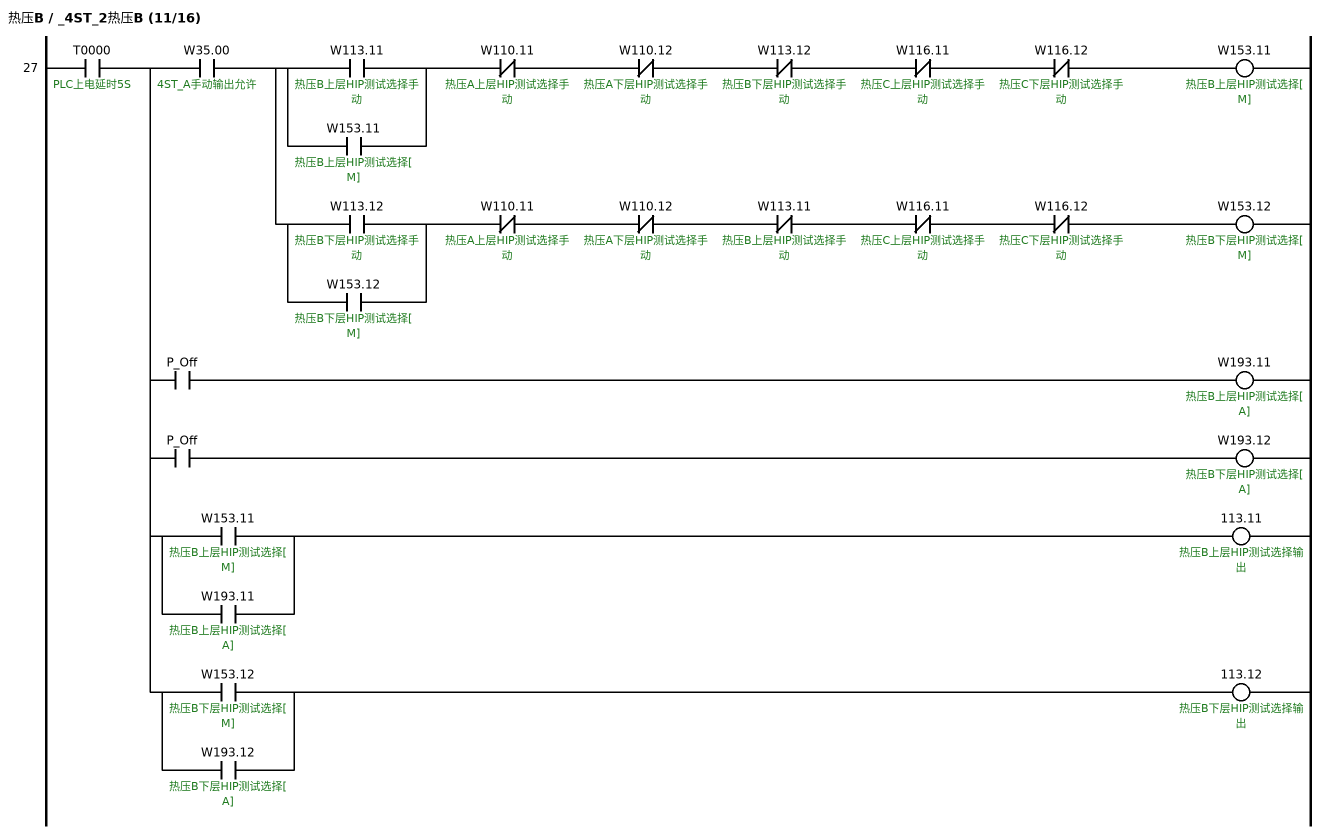
; [picture p192: 热压B / _4ST_2热压B, rungs 27-27]
; rung 27
LD T0000  ; PLC上电延时5S
OUT TR0
AND W35.00  ; 4ST_A手动输出允许
OUT TR1
LD W113.11  ; 热压B上层HIP测试选择手动
OR W153.11  ; 热压B上层HIP测试选择[M]
ANDLD
ANDNOT W110.11  ; 热压A上层HIP测试选择手动
ANDNOT W110.12  ; 热压A下层HIP测试选择手动
ANDNOT W113.12  ; 热压B下层HIP测试选择手动
ANDNOT W116.11  ; 热压C上层HIP测试选择手动
ANDNOT W116.12  ; 热压C下层HIP测试选择手动
OUT W153.11  ; 热压B上层HIP测试选择[M]
LD TR1
LD W113.12  ; 热压B下层HIP测试选择手动
OR W153.12  ; 热压B下层HIP测试选择[M]
ANDLD
ANDNOT W110.11  ; 热压A上层HIP测试选择手动
ANDNOT W110.12  ; 热压A下层HIP测试选择手动
ANDNOT W113.11  ; 热压B上层HIP测试选择手动
ANDNOT W116.11  ; 热压C上层HIP测试选择手动
ANDNOT W116.12  ; 热压C下层HIP测试选择手动
OUT W153.12  ; 热压B下层HIP测试选择[M]
LD TR0
AND P_Off
OUT W193.11  ; 热压B上层HIP测试选择[A]
LD TR0
AND P_Off
OUT W193.12  ; 热压B下层HIP测试选择[A]
LD TR0
LD W153.11  ; 热压B上层HIP测试选择[M]
OR W193.11  ; 热压B上层HIP测试选择[A]
ANDLD
OUT 113.11  ; 热压B上层HIP测试选择输出
LD TR0
LD W153.12  ; 热压B下层HIP测试选择[M]
OR W193.12  ; 热压B下层HIP测试选择[A]
ANDLD
OUT 113.12  ; 热压B下层HIP测试选择输出

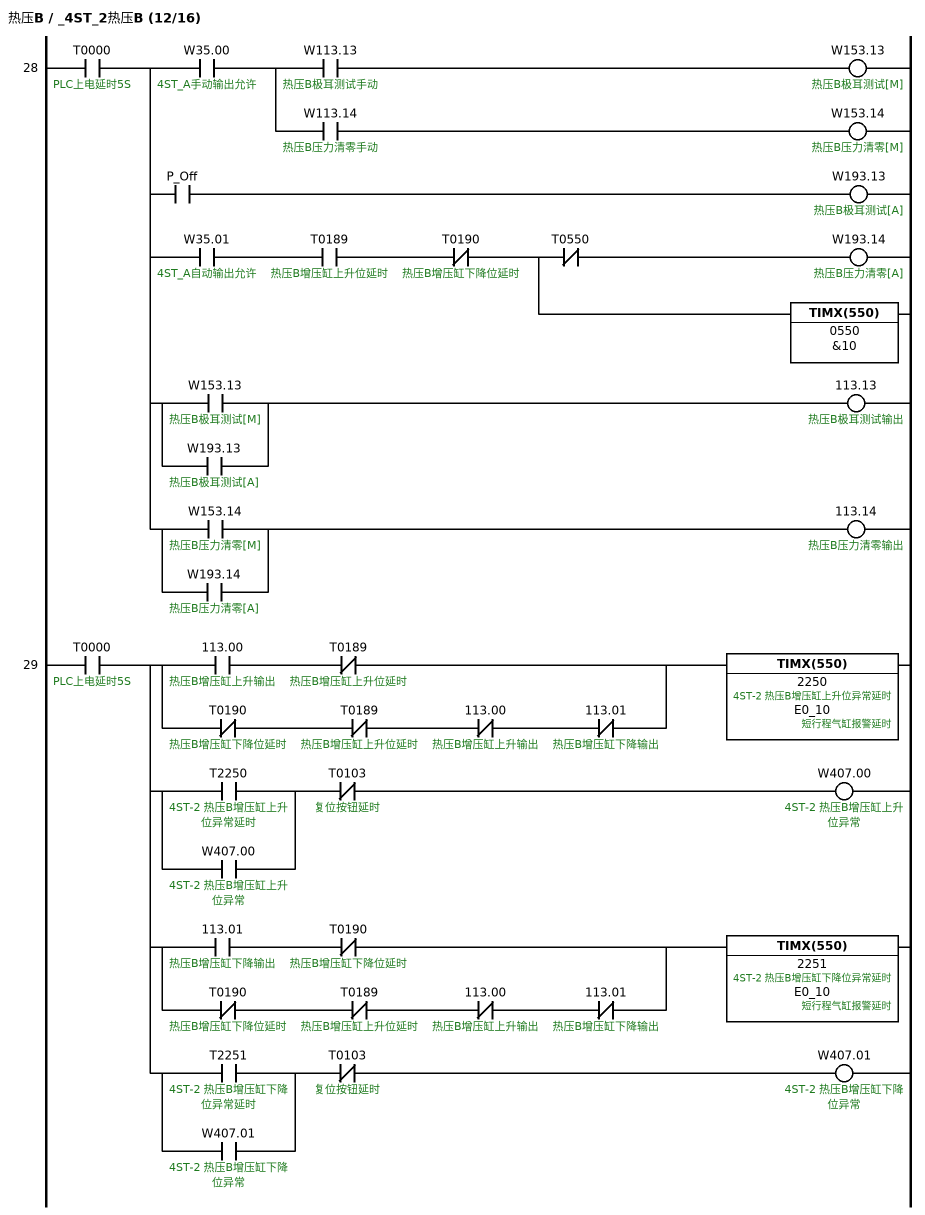
; rung 28
LD T0000  ; PLC上电延时5S
OUT TR0
AND W35.00  ; 4ST_A手动输出允许
OUT TR1
AND W113.13  ; 热压B极耳测试手动
OUT W153.13  ; 热压B极耳测试[M]
LD TR1
AND W113.14  ; 热压B压力清零手动
OUT W153.14  ; 热压B压力清零[M]
LD TR0
AND P_Off
OUT W193.13  ; 热压B极耳测试[A]
LD TR0
AND W35.01  ; 4ST_A自动输出允许
AND T0189  ; 热压B增压缸上升位延时
ANDNOT T0190  ; 热压B增压缸下降位延时
OUT TR1
ANDNOT T0550
OUT W193.14  ; 热压B压力清零[A]
LD TR1
TIMX(550) 0550 &10
LD TR0
LD W153.13  ; 热压B极耳测试[M]
OR W193.13  ; 热压B极耳测试[A]
ANDLD
OUT 113.13  ; 热压B极耳测试输出
LD TR0
LD W153.14  ; 热压B压力清零[M]
OR W193.14  ; 热压B压力清零[A]
ANDLD
OUT 113.14  ; 热压B压力清零输出
; rung 29
LD T0000  ; PLC上电延时5S
OUT TR0
LD 113.00  ; 热压B增压缸上升输出
ANDNOT T0189  ; 热压B增压缸上升位延时
LDNOT T0190  ; 热压B增压缸下降位延时
ANDNOT T0189  ; 热压B增压缸上升位延时
ANDNOT 113.00  ; 热压B增压缸上升输出
ANDNOT 113.01  ; 热压B增压缸下降输出
ORLD
ANDLD
TIMX(550) 2250 E0_10  ; 短行程气缸报警延时, 4ST-2 热压B增压缸上升位异常延时
LD TR0
LD T2250  ; 4ST-2 热压B增压缸上升位异常延时
OR W407.00  ; 4ST-2 热压B增压缸上升位异常
ANDLD
ANDNOT T0103  ; 复位按钮延时
OUT W407.00  ; 4ST-2 热压B增压缸上升位异常
LD TR0
LD 113.01  ; 热压B增压缸下降输出
ANDNOT T0190  ; 热压B增压缸下降位延时
LDNOT T0190  ; 热压B增压缸下降位延时
ANDNOT T0189  ; 热压B增压缸上升位延时
ANDNOT 113.00  ; 热压B增压缸上升输出
ANDNOT 113.01  ; 热压B增压缸下降输出
ORLD
ANDLD
TIMX(550) 2251 E0_10  ; 短行程气缸报警延时, 4ST-2 热压B增压缸下降位异常延时
LD TR0
LD T2251  ; 4ST-2 热压B增压缸下降位异常延时
OR W407.01  ; 4ST-2 热压B增压缸下降位异常
ANDLD
ANDNOT T0103  ; 复位按钮延时
OUT W407.01  ; 4ST-2 热压B增压缸下降位异常

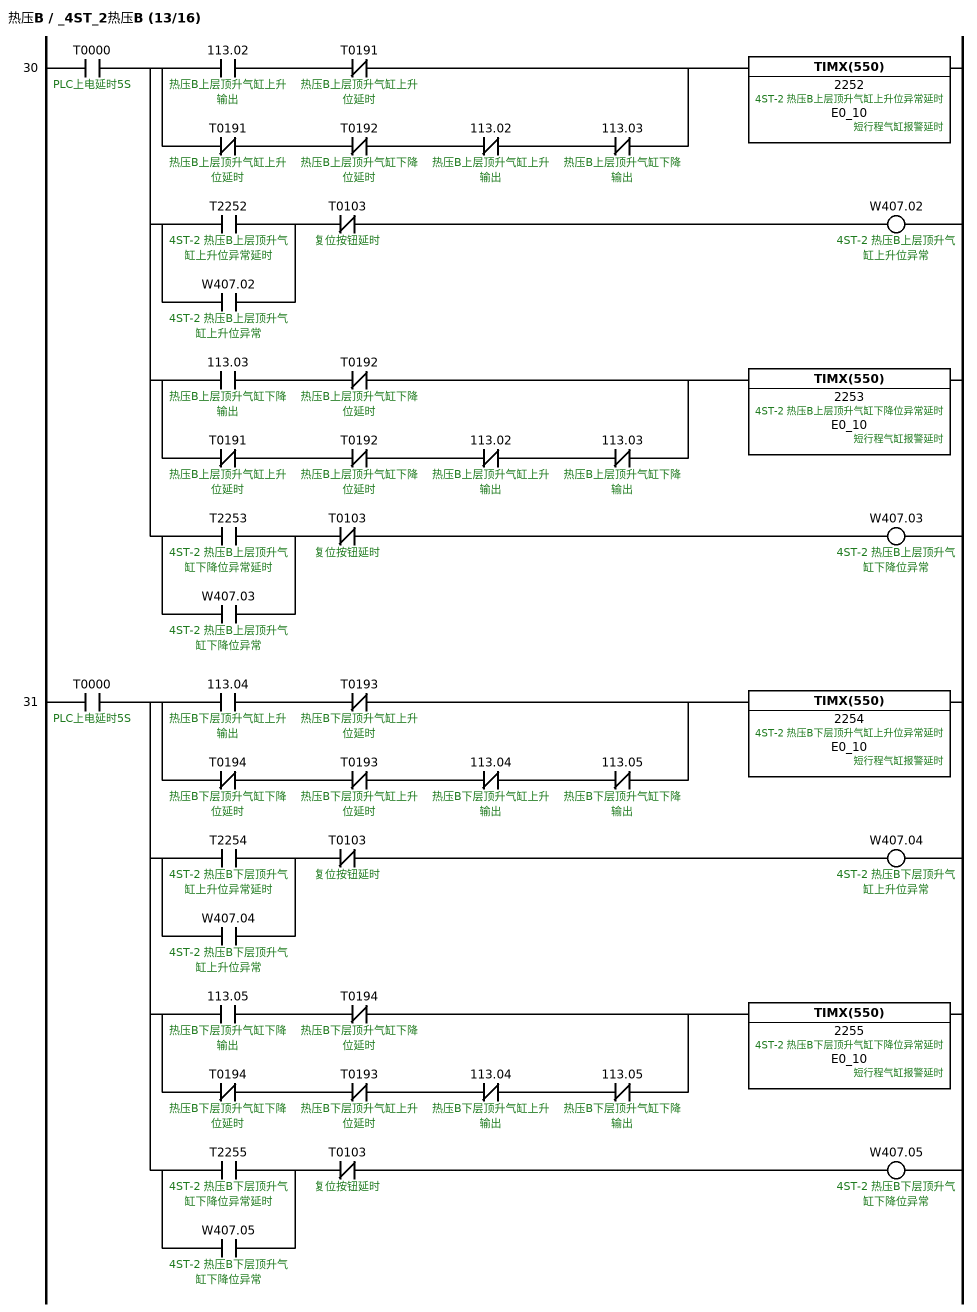
; rung 30
LD T0000  ; PLC上电延时5S
OUT TR0
LD 113.02  ; 热压B上层顶升气缸上升输出
ANDNOT T0191  ; 热压B上层顶升气缸上升位延时
LDNOT T0191  ; 热压B上层顶升气缸上升位延时
ANDNOT T0192  ; 热压B上层顶升气缸下降位延时
ANDNOT 113.02  ; 热压B上层顶升气缸上升输出
ANDNOT 113.03  ; 热压B上层顶升气缸下降输出
ORLD
ANDLD
TIMX(550) 2252 E0_10  ; 短行程气缸报警延时, 4ST-2 热压B上层顶升气缸上升位异常延时
LD TR0
LD T2252  ; 4ST-2 热压B上层顶升气缸上升位异常延时
OR W407.02  ; 4ST-2 热压B上层顶升气缸上升位异常
ANDLD
ANDNOT T0103  ; 复位按钮延时
OUT W407.02  ; 4ST-2 热压B上层顶升气缸上升位异常
LD TR0
LD 113.03  ; 热压B上层顶升气缸下降输出
ANDNOT T0192  ; 热压B上层顶升气缸下降位延时
LDNOT T0191  ; 热压B上层顶升气缸上升位延时
ANDNOT T0192  ; 热压B上层顶升气缸下降位延时
ANDNOT 113.02  ; 热压B上层顶升气缸上升输出
ANDNOT 113.03  ; 热压B上层顶升气缸下降输出
ORLD
ANDLD
TIMX(550) 2253 E0_10  ; 短行程气缸报警延时, 4ST-2 热压B上层顶升气缸下降位异常延时
LD TR0
LD T2253  ; 4ST-2 热压B上层顶升气缸下降位异常延时
OR W407.03  ; 4ST-2 热压B上层顶升气缸下降位异常
ANDLD
ANDNOT T0103  ; 复位按钮延时
OUT W407.03  ; 4ST-2 热压B上层顶升气缸下降位异常
; rung 31
LD T0000  ; PLC上电延时5S
OUT TR0
LD 113.04  ; 热压B下层顶升气缸上升输出
ANDNOT T0193  ; 热压B下层顶升气缸上升位延时
LDNOT T0194  ; 热压B下层顶升气缸下降位延时
ANDNOT T0193  ; 热压B下层顶升气缸上升位延时
ANDNOT 113.04  ; 热压B下层顶升气缸上升输出
ANDNOT 113.05  ; 热压B下层顶升气缸下降输出
ORLD
ANDLD
TIMX(550) 2254 E0_10  ; 短行程气缸报警延时, 4ST-2 热压B下层顶升气缸上升位异常延时
LD TR0
LD T2254  ; 4ST-2 热压B下层顶升气缸上升位异常延时
OR W407.04  ; 4ST-2 热压B下层顶升气缸上升位异常
ANDLD
ANDNOT T0103  ; 复位按钮延时
OUT W407.04  ; 4ST-2 热压B下层顶升气缸上升位异常
LD TR0
LD 113.05  ; 热压B下层顶升气缸下降输出
ANDNOT T0194  ; 热压B下层顶升气缸下降位延时
LDNOT T0194  ; 热压B下层顶升气缸下降位延时
ANDNOT T0193  ; 热压B下层顶升气缸上升位延时
ANDNOT 113.04  ; 热压B下层顶升气缸上升输出
ANDNOT 113.05  ; 热压B下层顶升气缸下降输出
ORLD
ANDLD
TIMX(550) 2255 E0_10  ; 短行程气缸报警延时, 4ST-2 热压B下层顶升气缸下降位异常延时
LD TR0
LD T2255  ; 4ST-2 热压B下层顶升气缸下降位异常延时
OR W407.05  ; 4ST-2 热压B下层顶升气缸下降位异常
ANDLD
ANDNOT T0103  ; 复位按钮延时
OUT W407.05  ; 4ST-2 热压B下层顶升气缸下降位异常

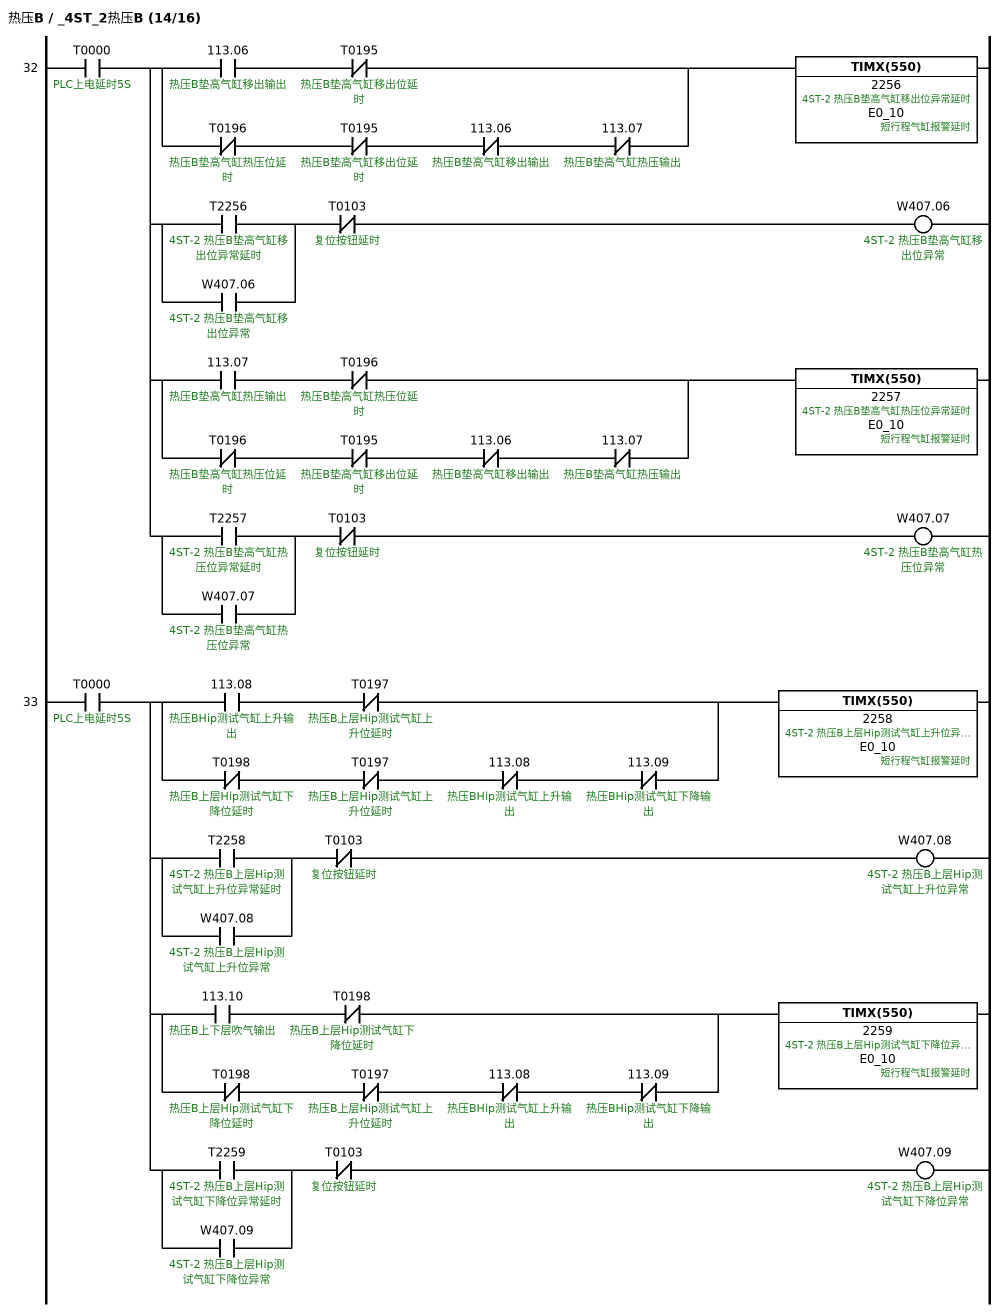
; rung 32
LD T0000  ; PLC上电延时5S
OUT TR0
LD 113.06  ; 热压B垫高气缸移出输出
ANDNOT T0195  ; 热压B垫高气缸移出位延时
LDNOT T0196  ; 热压B垫高气缸热压位延时
ANDNOT T0195  ; 热压B垫高气缸移出位延时
ANDNOT 113.06  ; 热压B垫高气缸移出输出
ANDNOT 113.07  ; 热压B垫高气缸热压输出
ORLD
ANDLD
TIMX(550) 2256 E0_10  ; 短行程气缸报警延时, 4ST-2 热压B垫高气缸移出位异常延时
LD TR0
LD T2256  ; 4ST-2 热压B垫高气缸移出位异常延时
OR W407.06  ; 4ST-2 热压B垫高气缸移出位异常
ANDLD
ANDNOT T0103  ; 复位按钮延时
OUT W407.06  ; 4ST-2 热压B垫高气缸移出位异常
LD TR0
LD 113.07  ; 热压B垫高气缸热压输出
ANDNOT T0196  ; 热压B垫高气缸热压位延时
LDNOT T0196  ; 热压B垫高气缸热压位延时
ANDNOT T0195  ; 热压B垫高气缸移出位延时
ANDNOT 113.06  ; 热压B垫高气缸移出输出
ANDNOT 113.07  ; 热压B垫高气缸热压输出
ORLD
ANDLD
TIMX(550) 2257 E0_10  ; 短行程气缸报警延时, 4ST-2 热压B垫高气缸热压位异常延时
LD TR0
LD T2257  ; 4ST-2 热压B垫高气缸热压位异常延时
OR W407.07  ; 4ST-2 热压B垫高气缸热压位异常
ANDLD
ANDNOT T0103  ; 复位按钮延时
OUT W407.07  ; 4ST-2 热压B垫高气缸热压位异常
; rung 33
LD T0000  ; PLC上电延时5S
OUT TR0
LD 113.08  ; 热压BHip测试气缸上升输出
ANDNOT T0197  ; 热压B上层Hip测试气缸上升位延时
LDNOT T0198  ; 热压B上层Hip测试气缸下降位延时
ANDNOT T0197  ; 热压B上层Hip测试气缸上升位延时
ANDNOT 113.08  ; 热压BHip测试气缸上升输出
ANDNOT 113.09  ; 热压BHip测试气缸下降输出
ORLD
ANDLD
TIMX(550) 2258 E0_10  ; 短行程气缸报警延时, 4ST-2 热压B上层Hip测试气缸上升位异常延时
LD TR0
LD T2258  ; 4ST-2 热压B上层Hip测试气缸上升位异常延时
OR W407.08  ; 4ST-2 热压B上层Hip测试气缸上升位异常
ANDLD
ANDNOT T0103  ; 复位按钮延时
OUT W407.08  ; 4ST-2 热压B上层Hip测试气缸上升位异常
LD TR0
LD 113.10  ; 热压B上下层吹气输出
ANDNOT T0198  ; 热压B上层Hip测试气缸下降位延时
LDNOT T0198  ; 热压B上层Hip测试气缸下降位延时
ANDNOT T0197  ; 热压B上层Hip测试气缸上升位延时
ANDNOT 113.08  ; 热压BHip测试气缸上升输出
ANDNOT 113.09  ; 热压BHip测试气缸下降输出
ORLD
ANDLD
TIMX(550) 2259 E0_10  ; 短行程气缸报警延时, 4ST-2 热压B上层Hip测试气缸下降位异常延时
LD TR0
LD T2259  ; 4ST-2 热压B上层Hip测试气缸下降位异常延时
OR W407.09  ; 4ST-2 热压B上层Hip测试气缸下降位异常
ANDLD
ANDNOT T0103  ; 复位按钮延时
OUT W407.09  ; 4ST-2 热压B上层Hip测试气缸下降位异常

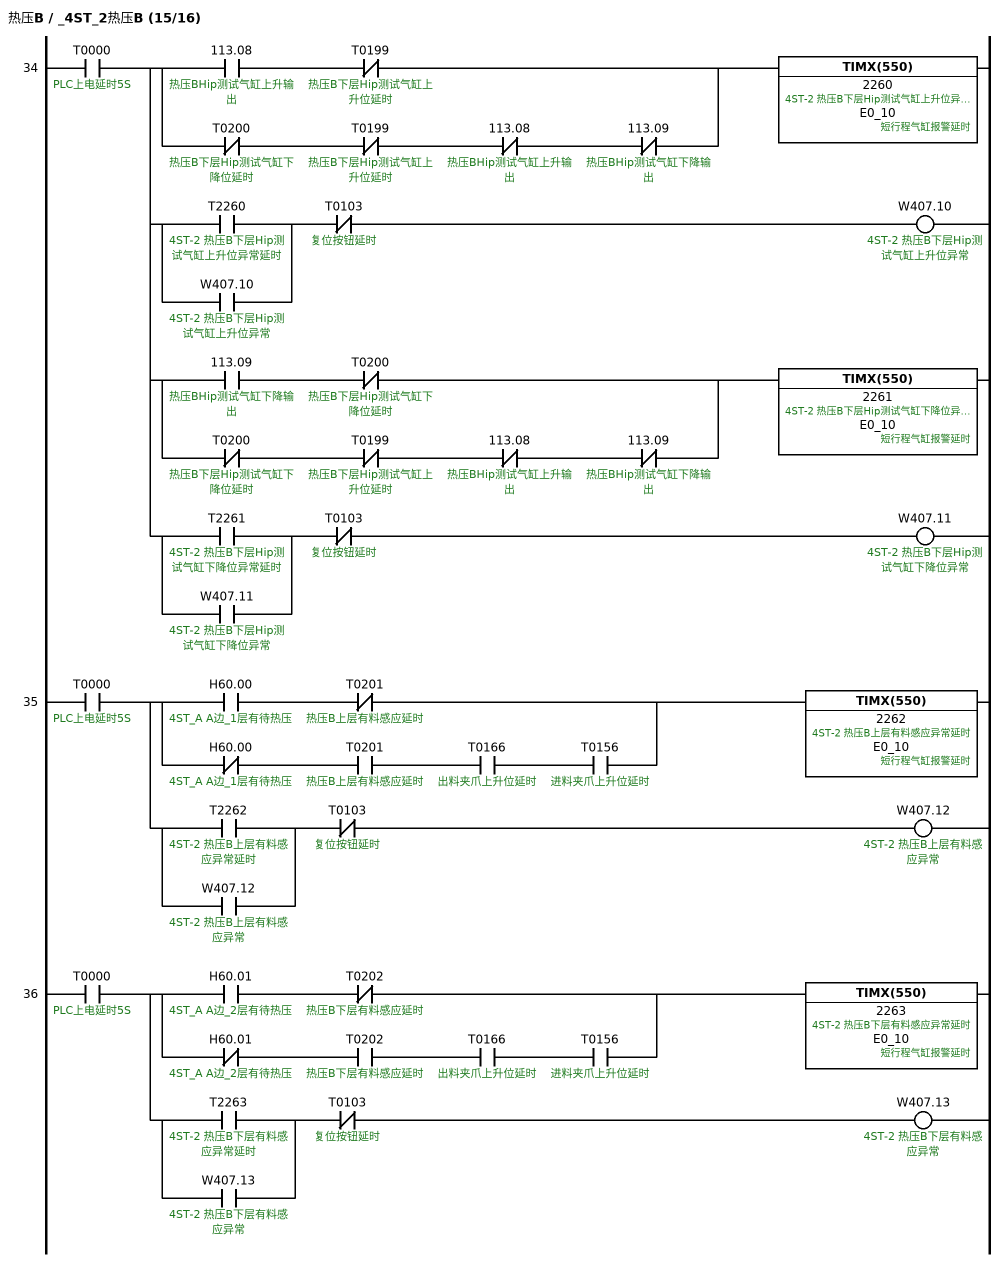
; rung 34
LD T0000  ; PLC上电延时5S
OUT TR0
LD 113.08  ; 热压BHip测试气缸上升输出
ANDNOT T0199  ; 热压B下层Hip测试气缸上升位延时
LDNOT T0200  ; 热压B下层Hip测试气缸下降位延时
ANDNOT T0199  ; 热压B下层Hip测试气缸上升位延时
ANDNOT 113.08  ; 热压BHip测试气缸上升输出
ANDNOT 113.09  ; 热压BHip测试气缸下降输出
ORLD
ANDLD
TIMX(550) 2260 E0_10  ; 短行程气缸报警延时, 4ST-2 热压B下层Hip测试气缸上升位异常延时
LD TR0
LD T2260  ; 4ST-2 热压B下层Hip测试气缸上升位异常延时
OR W407.10  ; 4ST-2 热压B下层Hip测试气缸上升位异常
ANDLD
ANDNOT T0103  ; 复位按钮延时
OUT W407.10  ; 4ST-2 热压B下层Hip测试气缸上升位异常
LD TR0
LD 113.09  ; 热压BHip测试气缸下降输出
ANDNOT T0200  ; 热压B下层Hip测试气缸下降位延时
LDNOT T0200  ; 热压B下层Hip测试气缸下降位延时
ANDNOT T0199  ; 热压B下层Hip测试气缸上升位延时
ANDNOT 113.08  ; 热压BHip测试气缸上升输出
ANDNOT 113.09  ; 热压BHip测试气缸下降输出
ORLD
ANDLD
TIMX(550) 2261 E0_10  ; 短行程气缸报警延时, 4ST-2 热压B下层Hip测试气缸下降位异常延时
LD TR0
LD T2261  ; 4ST-2 热压B下层Hip测试气缸下降位异常延时
OR W407.11  ; 4ST-2 热压B下层Hip测试气缸下降位异常
ANDLD
ANDNOT T0103  ; 复位按钮延时
OUT W407.11  ; 4ST-2 热压B下层Hip测试气缸下降位异常
; rung 35
LD T0000  ; PLC上电延时5S
OUT TR0
LD H60.00  ; 4ST_A A边_1层有待热压
ANDNOT T0201  ; 热压B上层有料感应延时
LDNOT H60.00  ; 4ST_A A边_1层有待热压
AND T0201  ; 热压B上层有料感应延时
AND T0166  ; 出料夹爪上升位延时
AND T0156  ; 进料夹爪上升位延时
ORLD
ANDLD
TIMX(550) 2262 E0_10  ; 短行程气缸报警延时, 4ST-2 热压B上层有料感应异常延时
LD TR0
LD T2262  ; 4ST-2 热压B上层有料感应异常延时
OR W407.12  ; 4ST-2 热压B上层有料感应异常
ANDLD
ANDNOT T0103  ; 复位按钮延时
OUT W407.12  ; 4ST-2 热压B上层有料感应异常
; rung 36
LD T0000  ; PLC上电延时5S
OUT TR0
LD H60.01  ; 4ST_A A边_2层有待热压
ANDNOT T0202  ; 热压B下层有料感应延时
LDNOT H60.01  ; 4ST_A A边_2层有待热压
AND T0202  ; 热压B下层有料感应延时
AND T0166  ; 出料夹爪上升位延时
AND T0156  ; 进料夹爪上升位延时
ORLD
ANDLD
TIMX(550) 2263 E0_10  ; 短行程气缸报警延时, 4ST-2 热压B下层有料感应异常延时
LD TR0
LD T2263  ; 4ST-2 热压B下层有料感应异常延时
OR W407.13  ; 4ST-2 热压B下层有料感应异常
ANDLD
ANDNOT T0103  ; 复位按钮延时
OUT W407.13  ; 4ST-2 热压B下层有料感应异常

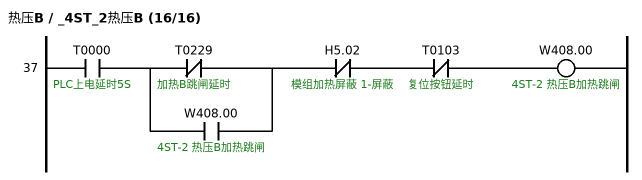
; rung 37
LD T0000  ; PLC上电延时5S
LDNOT T0229  ; 加热B跳闸延时
OR W408.00  ; 4ST-2 热压B加热跳闸
ANDLD
ANDNOT H5.02  ; 模组加热屏蔽 1-屏蔽
ANDNOT T0103  ; 复位按钮延时
OUT W408.00  ; 4ST-2 热压B加热跳闸

### Section 复位

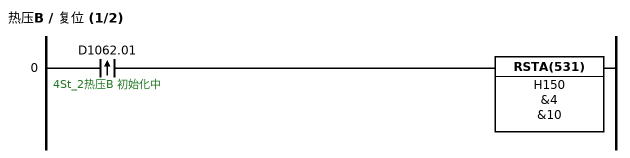
; rung 0
@LD D1062.01  ; 4St_2热压B 初始化中
RSTA(531) H150 &4 &10

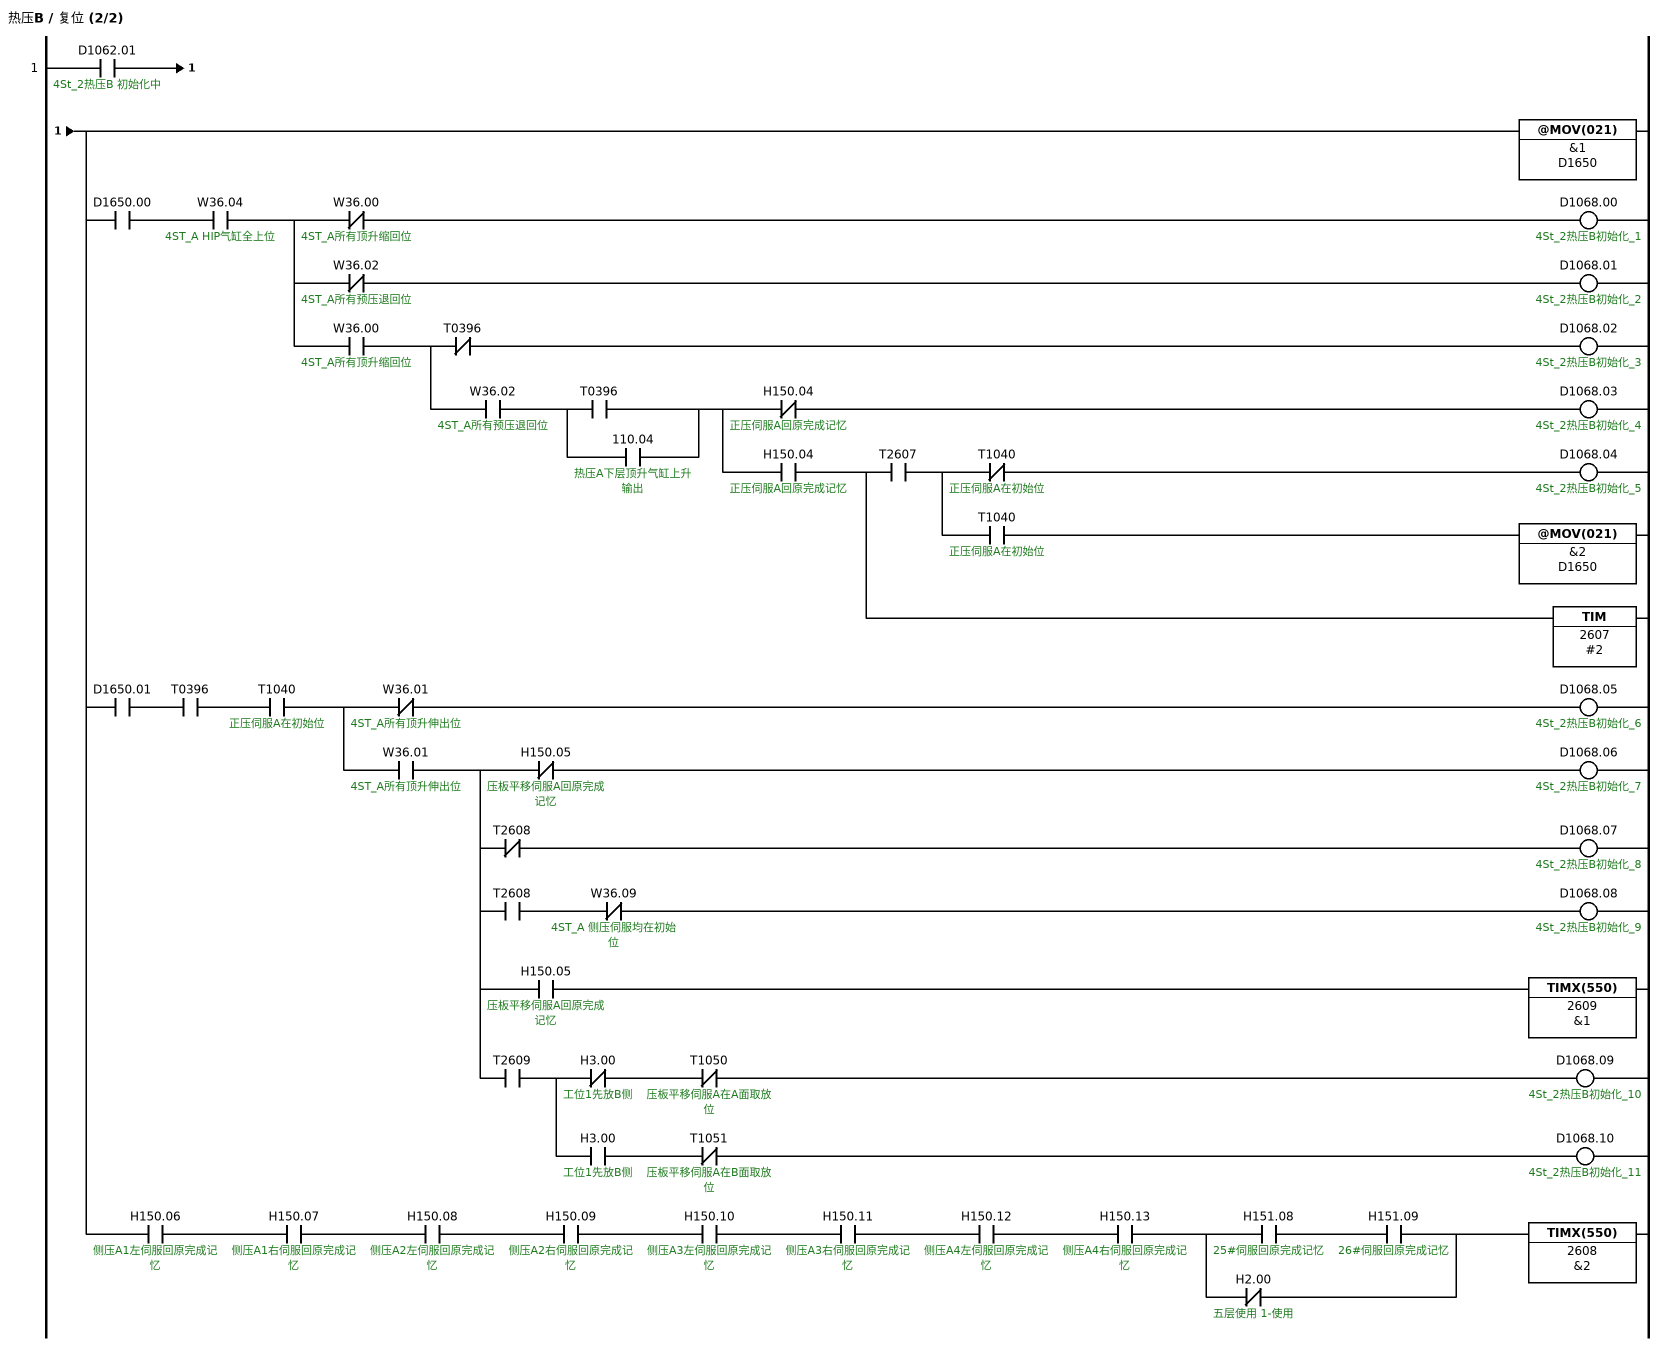
; rung 1
LD D1062.01  ; 4St_2热压B 初始化中
OUT TR0
@MOV(021) &1 D1650
AND D1650.00
AND W36.04  ; 4ST_A HIP气缸全上位
OUT TR1
ANDNOT W36.00  ; 4ST_A所有顶升缩回位
OUT D1068.00  ; 4St_2热压B初始化_1
LD TR1
ANDNOT W36.02  ; 4ST_A所有预压退回位
OUT D1068.01  ; 4St_2热压B初始化_2
LD TR1
AND W36.00  ; 4ST_A所有顶升缩回位
OUT TR1
ANDNOT T0396
OUT D1068.02  ; 4St_2热压B初始化_3
LD TR1
AND W36.02  ; 4ST_A所有预压退回位
LD T0396
OR 110.04  ; 热压A下层顶升气缸上升输出
ANDLD
OUT TR1
ANDNOT H150.04  ; 正压伺服A回原完成记忆
OUT D1068.03  ; 4St_2热压B初始化_4
LD TR1
AND H150.04  ; 正压伺服A回原完成记忆
OUT TR1
AND T2607
OUT TR2
ANDNOT T1040  ; 正压伺服A在初始位
OUT D1068.04  ; 4St_2热压B初始化_5
LD TR2
AND T1040  ; 正压伺服A在初始位
@MOV(021) &2 D1650
LD TR1
TIM 2607 #2
LD TR0
AND D1650.01
AND T0396
AND T1040  ; 正压伺服A在初始位
OUT TR1
ANDNOT W36.01  ; 4ST_A所有顶升伸出位
OUT D1068.05  ; 4St_2热压B初始化_6
LD TR1
AND W36.01  ; 4ST_A所有顶升伸出位
OUT TR1
ANDNOT H150.05  ; 压板平移伺服A回原完成记忆
OUT D1068.06  ; 4St_2热压B初始化_7
LD TR1
ANDNOT T2608
OUT D1068.07  ; 4St_2热压B初始化_8
LD TR1
AND T2608
ANDNOT W36.09  ; 4ST_A 侧压伺服均在初始位
OUT D1068.08  ; 4St_2热压B初始化_9
LD TR1
AND H150.05  ; 压板平移伺服A回原完成记忆
TIMX(550) 2609 &1
LD TR1
AND T2609
OUT TR1
ANDNOT H3.00  ; 工位1先放B侧
ANDNOT T1050  ; 压板平移伺服A在A面取放位
OUT D1068.09  ; 4St_2热压B初始化_10
LD TR1
AND H3.00  ; 工位1先放B侧
ANDNOT T1051  ; 压板平移伺服A在B面取放位
OUT D1068.10  ; 4St_2热压B初始化_11
LD TR0
AND H150.06  ; 侧压A1左伺服回原完成记忆
AND H150.07  ; 侧压A1右伺服回原完成记忆
AND H150.08  ; 侧压A2左伺服回原完成记忆
AND H150.09  ; 侧压A2右伺服回原完成记忆
AND H150.10  ; 侧压A3左伺服回原完成记忆
AND H150.11  ; 侧压A3右伺服回原完成记忆
AND H150.12  ; 侧压A4左伺服回原完成记忆
AND H150.13  ; 侧压A4右伺服回原完成记忆
LD H151.08  ; 25#伺服回原完成记忆
AND H151.09  ; 26#伺服回原完成记忆
ORNOT H2.00  ; 五层使用 1-使用
ANDLD
TIMX(550) 2608 &2

### Section 输出

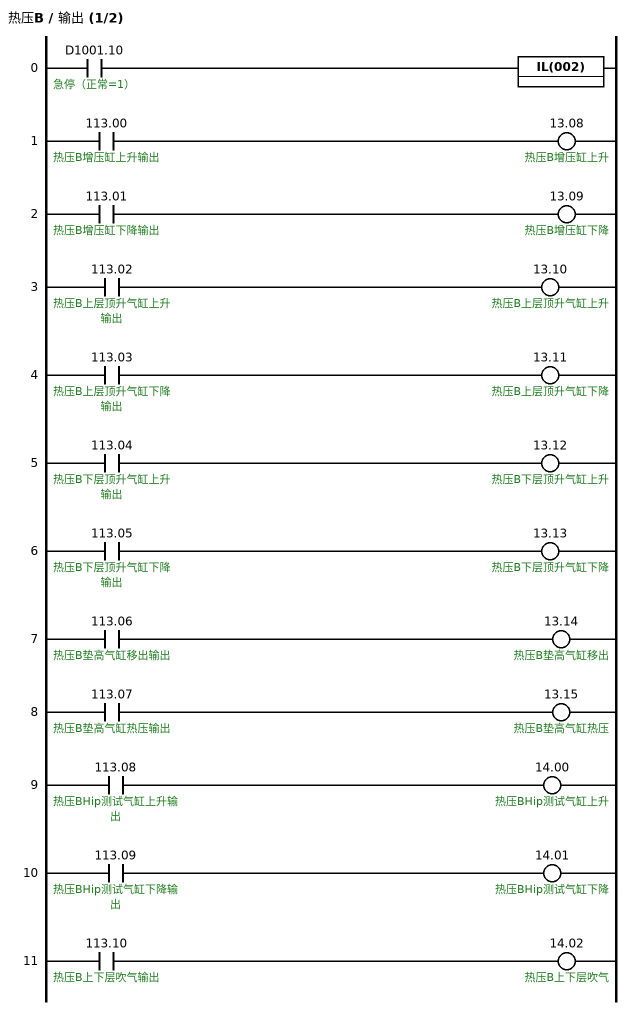
; rung 0
LD D1001.10  ; 急停（正常=1）
IL(002)
; rung 1
LD 113.00  ; 热压B增压缸上升输出
OUT 13.08  ; 热压B增压缸上升
; rung 2
LD 113.01  ; 热压B增压缸下降输出
OUT 13.09  ; 热压B增压缸下降
; rung 3
LD 113.02  ; 热压B上层顶升气缸上升输出
OUT 13.10  ; 热压B上层顶升气缸上升
; rung 4
LD 113.03  ; 热压B上层顶升气缸下降输出
OUT 13.11  ; 热压B上层顶升气缸下降
; rung 5
LD 113.04  ; 热压B下层顶升气缸上升输出
OUT 13.12  ; 热压B下层顶升气缸上升
; rung 6
LD 113.05  ; 热压B下层顶升气缸下降输出
OUT 13.13  ; 热压B下层顶升气缸下降
; rung 7
LD 113.06  ; 热压B垫高气缸移出输出
OUT 13.14  ; 热压B垫高气缸移出
; rung 8
LD 113.07  ; 热压B垫高气缸热压输出
OUT 13.15  ; 热压B垫高气缸热压
; rung 9
LD 113.08  ; 热压BHip测试气缸上升输出
OUT 14.00  ; 热压BHip测试气缸上升
; rung 10
LD 113.09  ; 热压BHip测试气缸下降输出
OUT 14.01  ; 热压BHip测试气缸下降
; rung 11
LD 113.10  ; 热压B上下层吹气输出
OUT 14.02  ; 热压B上下层吹气

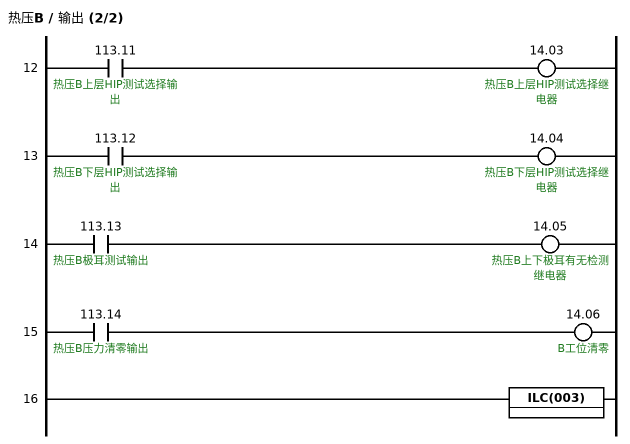
; rung 12
LD 113.11  ; 热压B上层HIP测试选择输出
OUT 14.03  ; 热压B上层HIP测试选择继电器
; rung 13
LD 113.12  ; 热压B下层HIP测试选择输出
OUT 14.04  ; 热压B下层HIP测试选择继电器
; rung 14
LD 113.13  ; 热压B极耳测试输出
OUT 14.05  ; 热压B上下极耳有无检测继电器
; rung 15
LD 113.14  ; 热压B压力清零输出
OUT 14.06  ; B工位清零
; rung 16
ILC(003)

### Section END
; rung 0
END(001)

## Program 热压C (cyclic task 6)

### Section Main

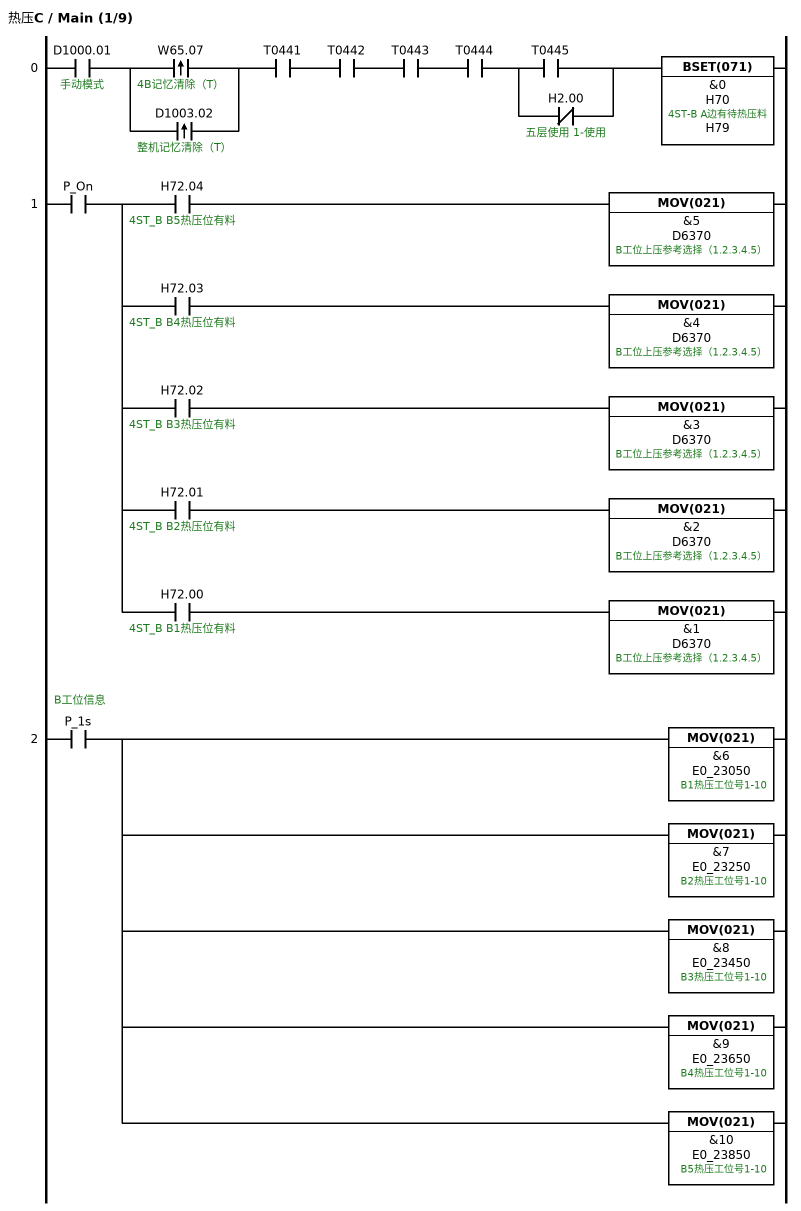
; rung 0
LD D1000.01  ; 手动模式
@LD W65.07  ; 4B记忆清除（T）
@OR D1003.02  ; 整机记忆清除（T）
ANDLD
AND T0441
AND T0442
AND T0443
AND T0444
LD T0445
ORNOT H2.00  ; 五层使用 1-使用
ANDLD
BSET(071) &0 H70 H79  ; 4ST-B A边有待热压料
; rung 1
LD P_On
OUT TR0
AND H72.04  ; 4ST_B B5热压位有料
MOV(021) &5 D6370  ; B工位上压参考选择（1.2.3.4.5）
LD TR0
AND H72.03  ; 4ST_B B4热压位有料
MOV(021) &4 D6370  ; B工位上压参考选择（1.2.3.4.5）
LD TR0
AND H72.02  ; 4ST_B B3热压位有料
MOV(021) &3 D6370  ; B工位上压参考选择（1.2.3.4.5）
LD TR0
AND H72.01  ; 4ST_B B2热压位有料
MOV(021) &2 D6370  ; B工位上压参考选择（1.2.3.4.5）
LD TR0
AND H72.00  ; 4ST_B B1热压位有料
MOV(021) &1 D6370  ; B工位上压参考选择（1.2.3.4.5）
; rung 2: B工位信息
LD P_1s
MOV(021) &6 E0_23050  ; B1热压工位号1-10
MOV(021) &7 E0_23250  ; B2热压工位号1-10
MOV(021) &8 E0_23450  ; B3热压工位号1-10
MOV(021) &9 E0_23650  ; B4热压工位号1-10
MOV(021) &10 E0_23850  ; B5热压工位号1-10

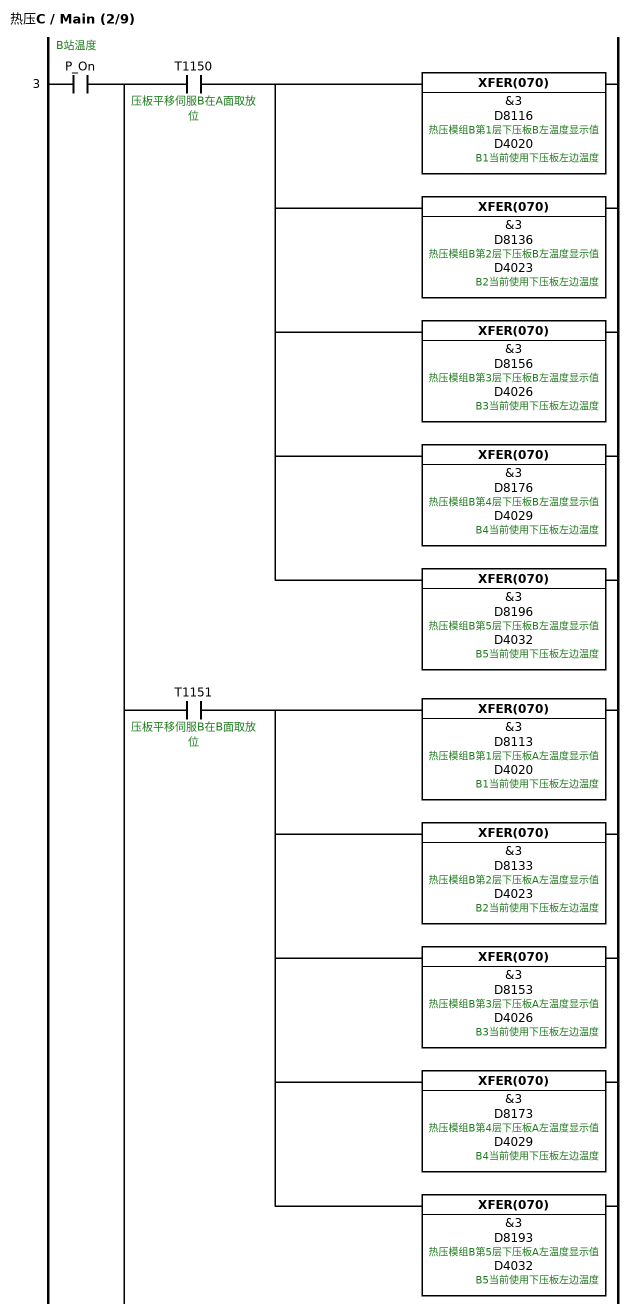

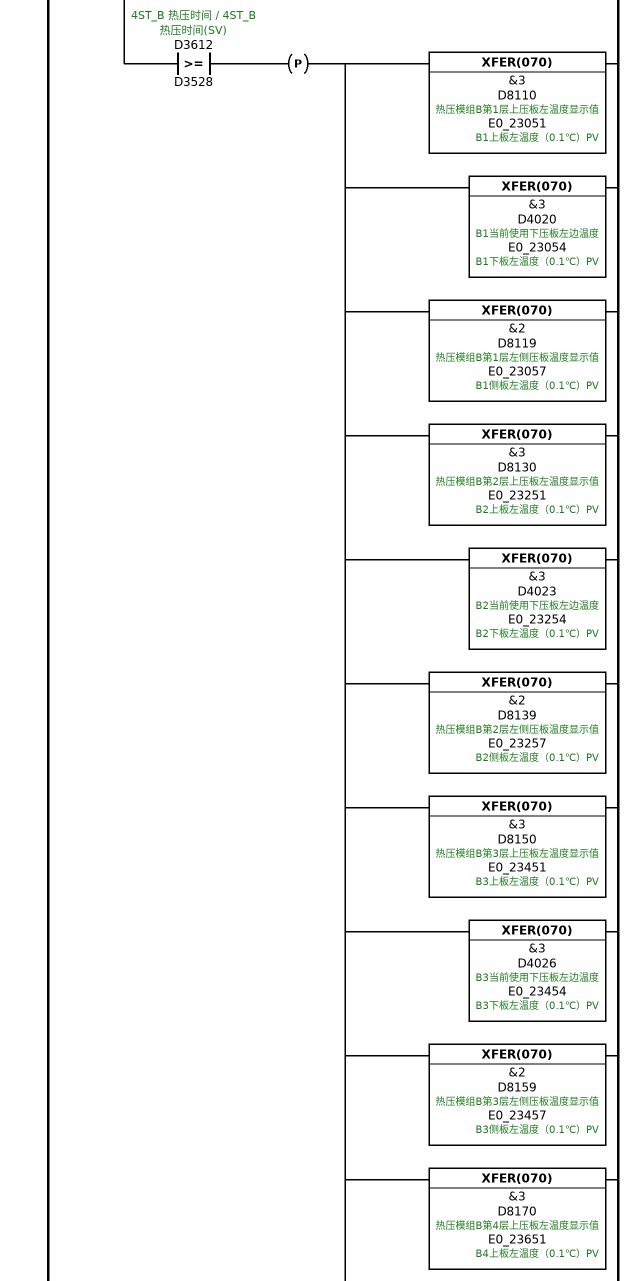

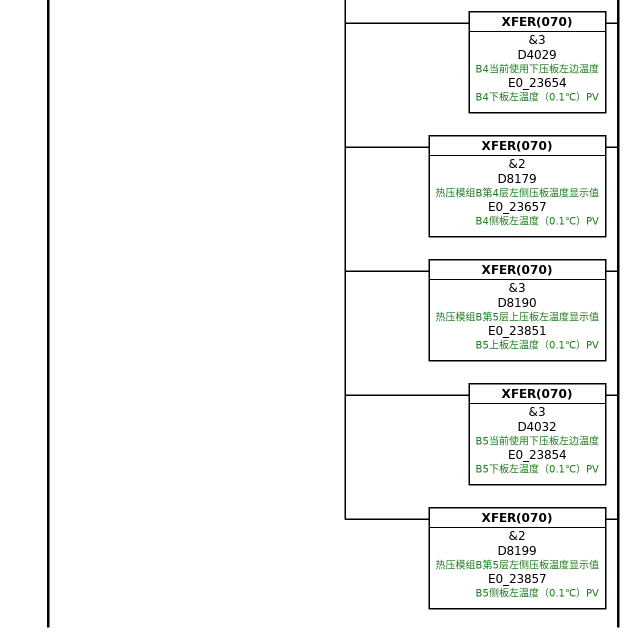
; rung 3: B站温度
LD P_On
OUT TR0
AND T1150  ; 压板平移伺服B在A面取放位
XFER(070) &3 D8116 D4020  ; 热压模组B第1层下压板B左温度显示值, B1当前使用下压板左边温度
XFER(070) &3 D8136 D4023  ; 热压模组B第2层下压板B左温度显示值, B2当前使用下压板左边温度
XFER(070) &3 D8156 D4026  ; 热压模组B第3层下压板B左温度显示值, B3当前使用下压板左边温度
XFER(070) &3 D8176 D4029  ; 热压模组B第4层下压板B左温度显示值, B4当前使用下压板左边温度
XFER(070) &3 D8196 D4032  ; 热压模组B第5层下压板B左温度显示值, B5当前使用下压板左边温度
LD TR0
AND T1151  ; 压板平移伺服B在B面取放位
XFER(070) &3 D8113 D4020  ; 热压模组B第1层下压板A左温度显示值, B1当前使用下压板左边温度
XFER(070) &3 D8133 D4023  ; 热压模组B第2层下压板A左温度显示值, B2当前使用下压板左边温度
XFER(070) &3 D8153 D4026  ; 热压模组B第3层下压板A左温度显示值, B3当前使用下压板左边温度
XFER(070) &3 D8173 D4029  ; 热压模组B第4层下压板A左温度显示值, B4当前使用下压板左边温度
XFER(070) &3 D8193 D4032  ; 热压模组B第5层下压板A左温度显示值, B5当前使用下压板左边温度
LD TR0
AND>=(325) D3612 D3528  ; 4ST_B 热压时间, 4ST_B 热压时间(SV)
UP(521)
XFER(070) &3 D8110 E0_23051  ; 热压模组B第1层上压板左温度显示值, B1上板左温度（0.1℃）PV
XFER(070) &3 D4020 E0_23054  ; B1当前使用下压板左边温度, B1下板左温度（0.1℃）PV
XFER(070) &2 D8119 E0_23057  ; 热压模组B第1层左侧压板温度显示值, B1侧板左温度（0.1℃）PV
XFER(070) &3 D8130 E0_23251  ; 热压模组B第2层上压板左温度显示值, B2上板左温度（0.1℃）PV
XFER(070) &3 D4023 E0_23254  ; B2当前使用下压板左边温度, B2下板左温度（0.1℃）PV
XFER(070) &2 D8139 E0_23257  ; 热压模组B第2层左侧压板温度显示值, B2侧板左温度（0.1℃）PV
XFER(070) &3 D8150 E0_23451  ; 热压模组B第3层上压板左温度显示值, B3上板左温度（0.1℃）PV
XFER(070) &3 D4026 E0_23454  ; B3当前使用下压板左边温度, B3下板左温度（0.1℃）PV
XFER(070) &2 D8159 E0_23457  ; 热压模组B第3层左侧压板温度显示值, B3侧板左温度（0.1℃）PV
XFER(070) &3 D8170 E0_23651  ; 热压模组B第4层上压板左温度显示值, B4上板左温度（0.1℃）PV
XFER(070) &3 D4029 E0_23654  ; B4当前使用下压板左边温度, B4下板左温度（0.1℃）PV
XFER(070) &2 D8179 E0_23657  ; 热压模组B第4层左侧压板温度显示值, B4侧板左温度（0.1℃）PV
XFER(070) &3 D8190 E0_23851  ; 热压模组B第5层上压板左温度显示值, B5上板左温度（0.1℃）PV
XFER(070) &3 D4032 E0_23854  ; B5当前使用下压板左边温度, B5下板左温度（0.1℃）PV
XFER(070) &2 D8199 E0_23857  ; 热压模组B第5层左侧压板温度显示值, B5侧板左温度（0.1℃）PV

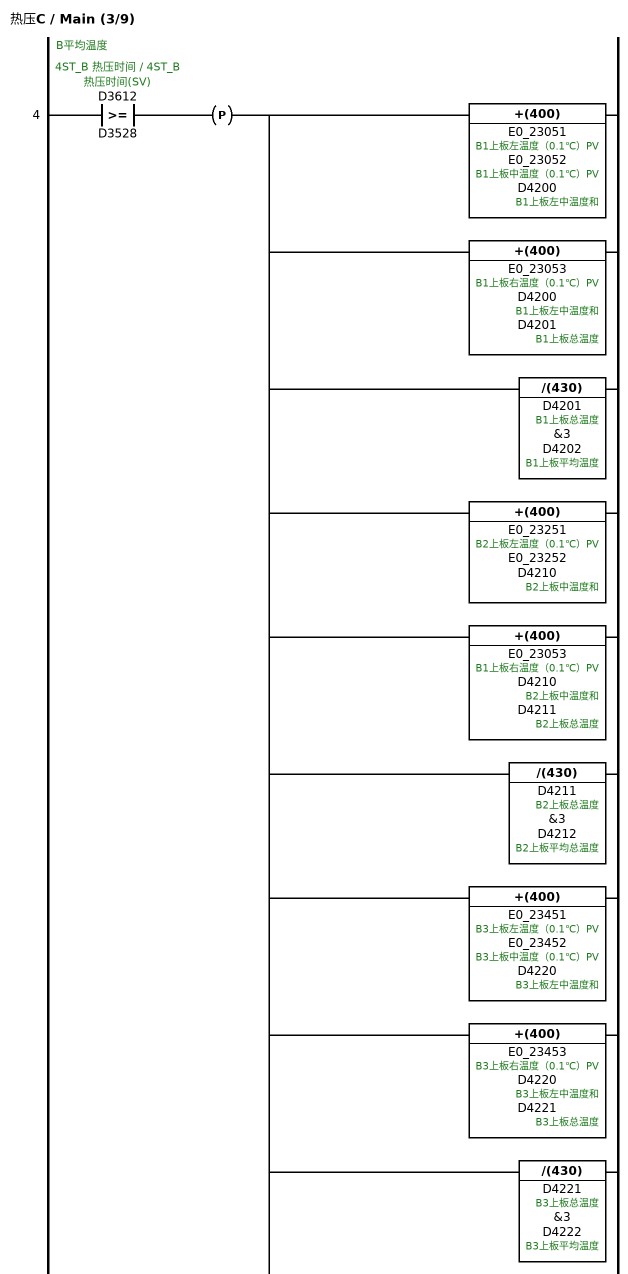

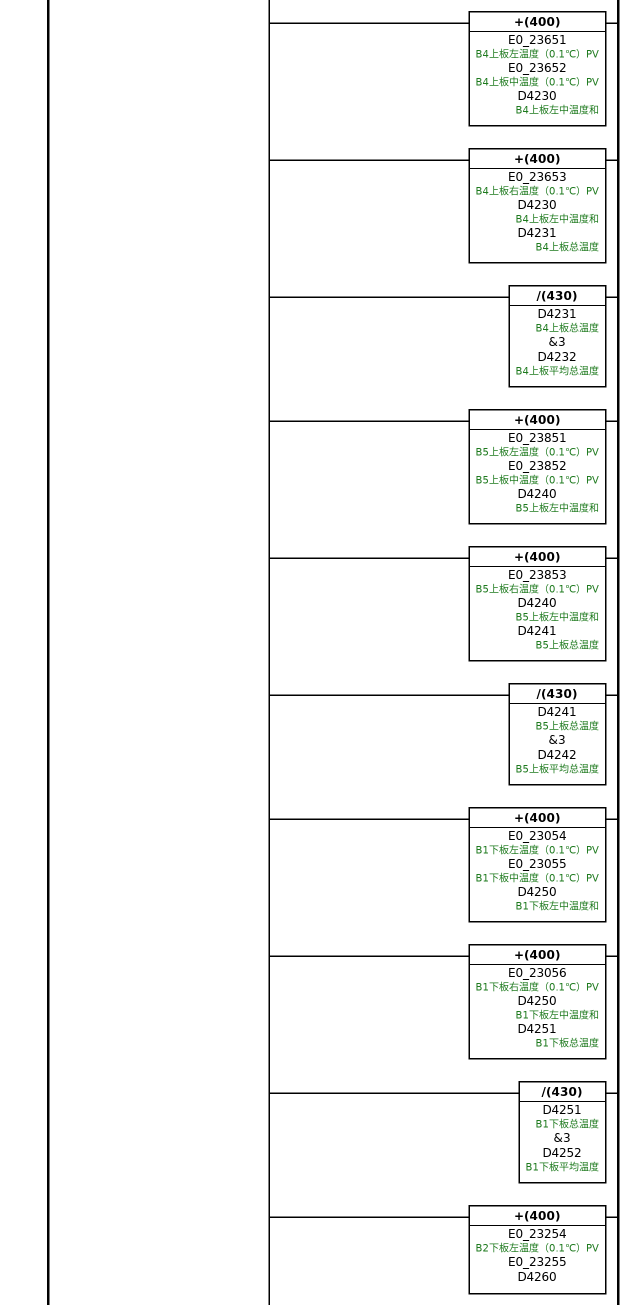

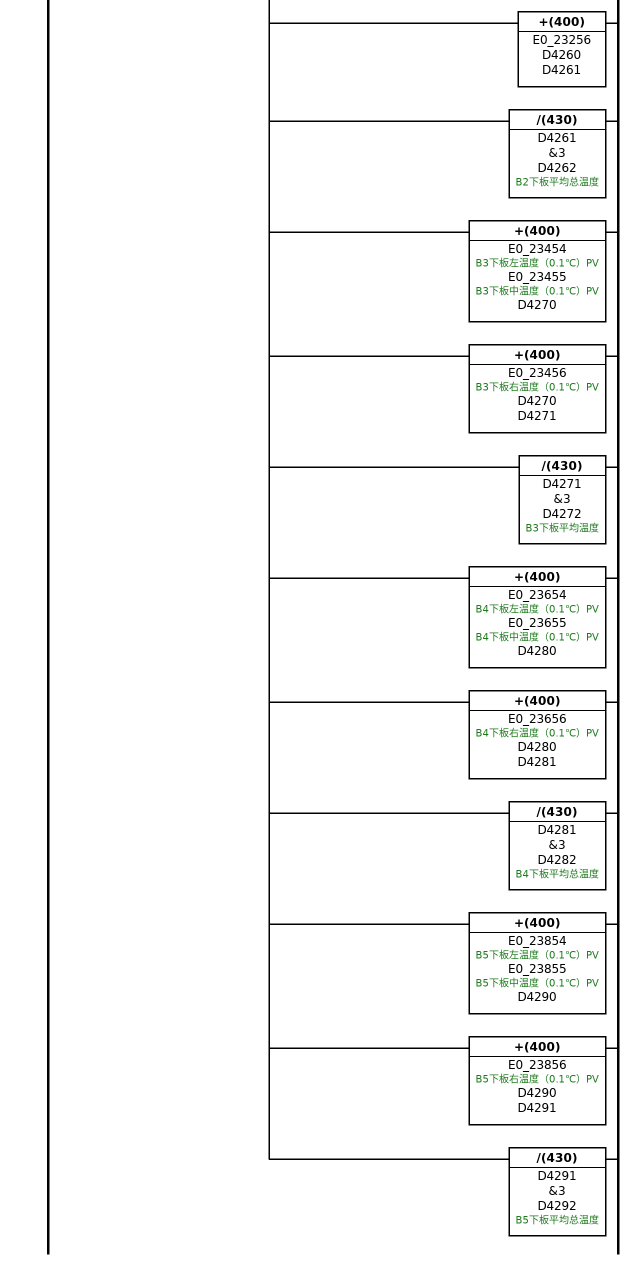
; rung 4: B平均温度
LD>=(325) D3612 D3528  ; 4ST_B 热压时间, 4ST_B 热压时间(SV)
UP(521)
+(400) E0_23051 E0_23052 D4200  ; B1上板左温度（0.1℃）PV, B1上板中温度（0.1℃）PV, B1上板左中温度和
+(400) E0_23053 D4200 D4201  ; B1上板右温度（0.1℃）PV, B1上板左中温度和, B1上板总温度
/(430) D4201 &3 D4202  ; B1上板总温度, B1上板平均温度
+(400) E0_23251 E0_23252 D4210  ; B2上板左温度（0.1℃）PV, B2上板中温度和
+(400) E0_23053 D4210 D4211  ; B1上板右温度（0.1℃）PV, B2上板中温度和, B2上板总温度
/(430) D4211 &3 D4212  ; B2上板总温度, B2上板平均总温度
+(400) E0_23451 E0_23452 D4220  ; B3上板左温度（0.1℃）PV, B3上板中温度（0.1℃）PV, B3上板左中温度和
+(400) E0_23453 D4220 D4221  ; B3上板右温度（0.1℃）PV, B3上板左中温度和, B3上板总温度
/(430) D4221 &3 D4222  ; B3上板总温度, B3上板平均温度
+(400) E0_23651 E0_23652 D4230  ; B4上板左温度（0.1℃）PV, B4上板中温度（0.1℃）PV, B4上板左中温度和
+(400) E0_23653 D4230 D4231  ; B4上板右温度（0.1℃）PV, B4上板左中温度和, B4上板总温度
/(430) D4231 &3 D4232  ; B4上板总温度, B4上板平均总温度
+(400) E0_23851 E0_23852 D4240  ; B5上板左温度（0.1℃）PV, B5上板中温度（0.1℃）PV, B5上板左中温度和
+(400) E0_23853 D4240 D4241  ; B5上板右温度（0.1℃）PV, B5上板左中温度和, B5上板总温度
/(430) D4241 &3 D4242  ; B5上板总温度, B5上板平均总温度
+(400) E0_23054 E0_23055 D4250  ; B1下板左温度（0.1℃）PV, B1下板中温度（0.1℃）PV, B1下板左中温度和
+(400) E0_23056 D4250 D4251  ; B1下板右温度（0.1℃）PV, B1下板左中温度和, B1下板总温度
/(430) D4251 &3 D4252  ; B1下板总温度, B1下板平均温度
+(400) E0_23254 E0_23255 D4260  ; B2下板左温度（0.1℃）PV
+(400) E0_23256 D4260 D4261
/(430) D4261 &3 D4262  ; B2下板平均总温度
+(400) E0_23454 E0_23455 D4270  ; B3下板左温度（0.1℃）PV, B3下板中温度（0.1℃）PV
+(400) E0_23456 D4270 D4271  ; B3下板右温度（0.1℃）PV
/(430) D4271 &3 D4272  ; B3下板平均温度
+(400) E0_23654 E0_23655 D4280  ; B4下板左温度（0.1℃）PV, B4下板中温度（0.1℃）PV
+(400) E0_23656 D4280 D4281  ; B4下板右温度（0.1℃）PV
/(430) D4281 &3 D4282  ; B4下板平均总温度
+(400) E0_23854 E0_23855 D4290  ; B5下板左温度（0.1℃）PV, B5下板中温度（0.1℃）PV
+(400) E0_23856 D4290 D4291  ; B5下板右温度（0.1℃）PV
/(430) D4291 &3 D4292  ; B5下板平均总温度

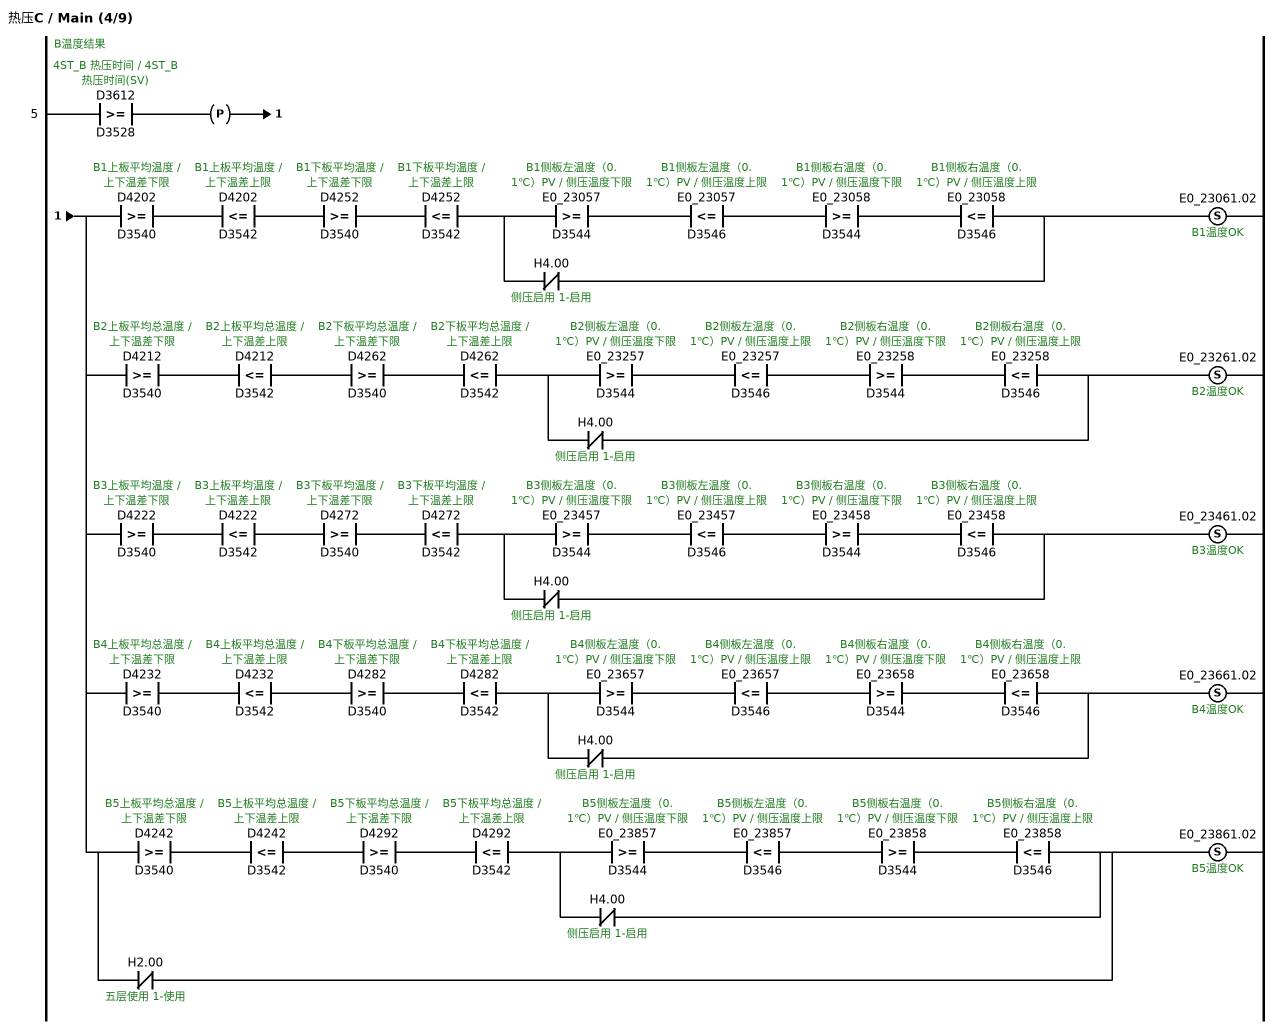
; rung 5: B温度结果
LD>=(325) D3612 D3528  ; 4ST_B 热压时间, 4ST_B 热压时间(SV)
UP(521)
OUT TR0
AND>=(325) D4202 D3540  ; B1上板平均温度, 上下温差下限
AND<=(315) D4202 D3542  ; B1上板平均温度, 上下温差上限
AND>=(325) D4252 D3540  ; B1下板平均温度, 上下温差下限
AND<=(315) D4252 D3542  ; B1下板平均温度, 上下温差上限
LD>=(325) E0_23057 D3544  ; B1侧板左温度（0.1℃）PV, 侧压温度下限
AND<=(315) E0_23057 D3546  ; B1侧板左温度（0.1℃）PV, 侧压温度上限
AND>=(325) E0_23058 D3544  ; B1侧板右温度（0.1℃）PV, 侧压温度下限
AND<=(315) E0_23058 D3546  ; B1侧板右温度（0.1℃）PV, 侧压温度上限
ORNOT H4.00  ; 侧压启用 1-启用
ANDLD
SET E0_23061.02  ; B1温度OK
LD TR0
AND>=(325) D4212 D3540  ; B2上板平均总温度, 上下温差下限
AND<=(315) D4212 D3542  ; B2上板平均总温度, 上下温差上限
AND>=(325) D4262 D3540  ; B2下板平均总温度, 上下温差下限
AND<=(315) D4262 D3542  ; B2下板平均总温度, 上下温差上限
LD>=(325) E0_23257 D3544  ; B2侧板左温度（0.1℃）PV, 侧压温度下限
AND<=(315) E0_23257 D3546  ; B2侧板左温度（0.1℃）PV, 侧压温度上限
AND>=(325) E0_23258 D3544  ; B2侧板右温度（0.1℃）PV, 侧压温度下限
AND<=(315) E0_23258 D3546  ; B2侧板右温度（0.1℃）PV, 侧压温度上限
ORNOT H4.00  ; 侧压启用 1-启用
ANDLD
SET E0_23261.02  ; B2温度OK
LD TR0
AND>=(325) D4222 D3540  ; B3上板平均温度, 上下温差下限
AND<=(315) D4222 D3542  ; B3上板平均温度, 上下温差上限
AND>=(325) D4272 D3540  ; B3下板平均温度, 上下温差下限
AND<=(315) D4272 D3542  ; B3下板平均温度, 上下温差上限
LD>=(325) E0_23457 D3544  ; B3侧板左温度（0.1℃）PV, 侧压温度下限
AND<=(315) E0_23457 D3546  ; B3侧板左温度（0.1℃）PV, 侧压温度上限
AND>=(325) E0_23458 D3544  ; B3侧板右温度（0.1℃）PV, 侧压温度下限
AND<=(315) E0_23458 D3546  ; B3侧板右温度（0.1℃）PV, 侧压温度上限
ORNOT H4.00  ; 侧压启用 1-启用
ANDLD
SET E0_23461.02  ; B3温度OK
LD TR0
AND>=(325) D4232 D3540  ; B4上板平均总温度, 上下温差下限
AND<=(315) D4232 D3542  ; B4上板平均总温度, 上下温差上限
AND>=(325) D4282 D3540  ; B4下板平均总温度, 上下温差下限
AND<=(315) D4282 D3542  ; B4下板平均总温度, 上下温差上限
LD>=(325) E0_23657 D3544  ; B4侧板左温度（0.1℃）PV, 侧压温度下限
AND<=(315) E0_23657 D3546  ; B4侧板左温度（0.1℃）PV, 侧压温度上限
AND>=(325) E0_23658 D3544  ; B4侧板右温度（0.1℃）PV, 侧压温度下限
AND<=(315) E0_23658 D3546  ; B4侧板右温度（0.1℃）PV, 侧压温度上限
ORNOT H4.00  ; 侧压启用 1-启用
ANDLD
SET E0_23661.02  ; B4温度OK
LD TR0
LD>=(325) D4242 D3540  ; B5上板平均总温度, 上下温差下限
AND<=(315) D4242 D3542  ; B5上板平均总温度, 上下温差上限
AND>=(325) D4292 D3540  ; B5下板平均总温度, 上下温差下限
AND<=(315) D4292 D3542  ; B5下板平均总温度, 上下温差上限
LD>=(325) E0_23857 D3544  ; B5侧板左温度（0.1℃）PV, 侧压温度下限
AND<=(315) E0_23857 D3546  ; B5侧板左温度（0.1℃）PV, 侧压温度上限
AND>=(325) E0_23858 D3544  ; B5侧板右温度（0.1℃）PV, 侧压温度下限
AND<=(315) E0_23858 D3546  ; B5侧板右温度（0.1℃）PV, 侧压温度上限
ORNOT H4.00  ; 侧压启用 1-启用
ANDLD
ORNOT H2.00  ; 五层使用 1-使用
ANDLD
SET E0_23861.02  ; B5温度OK

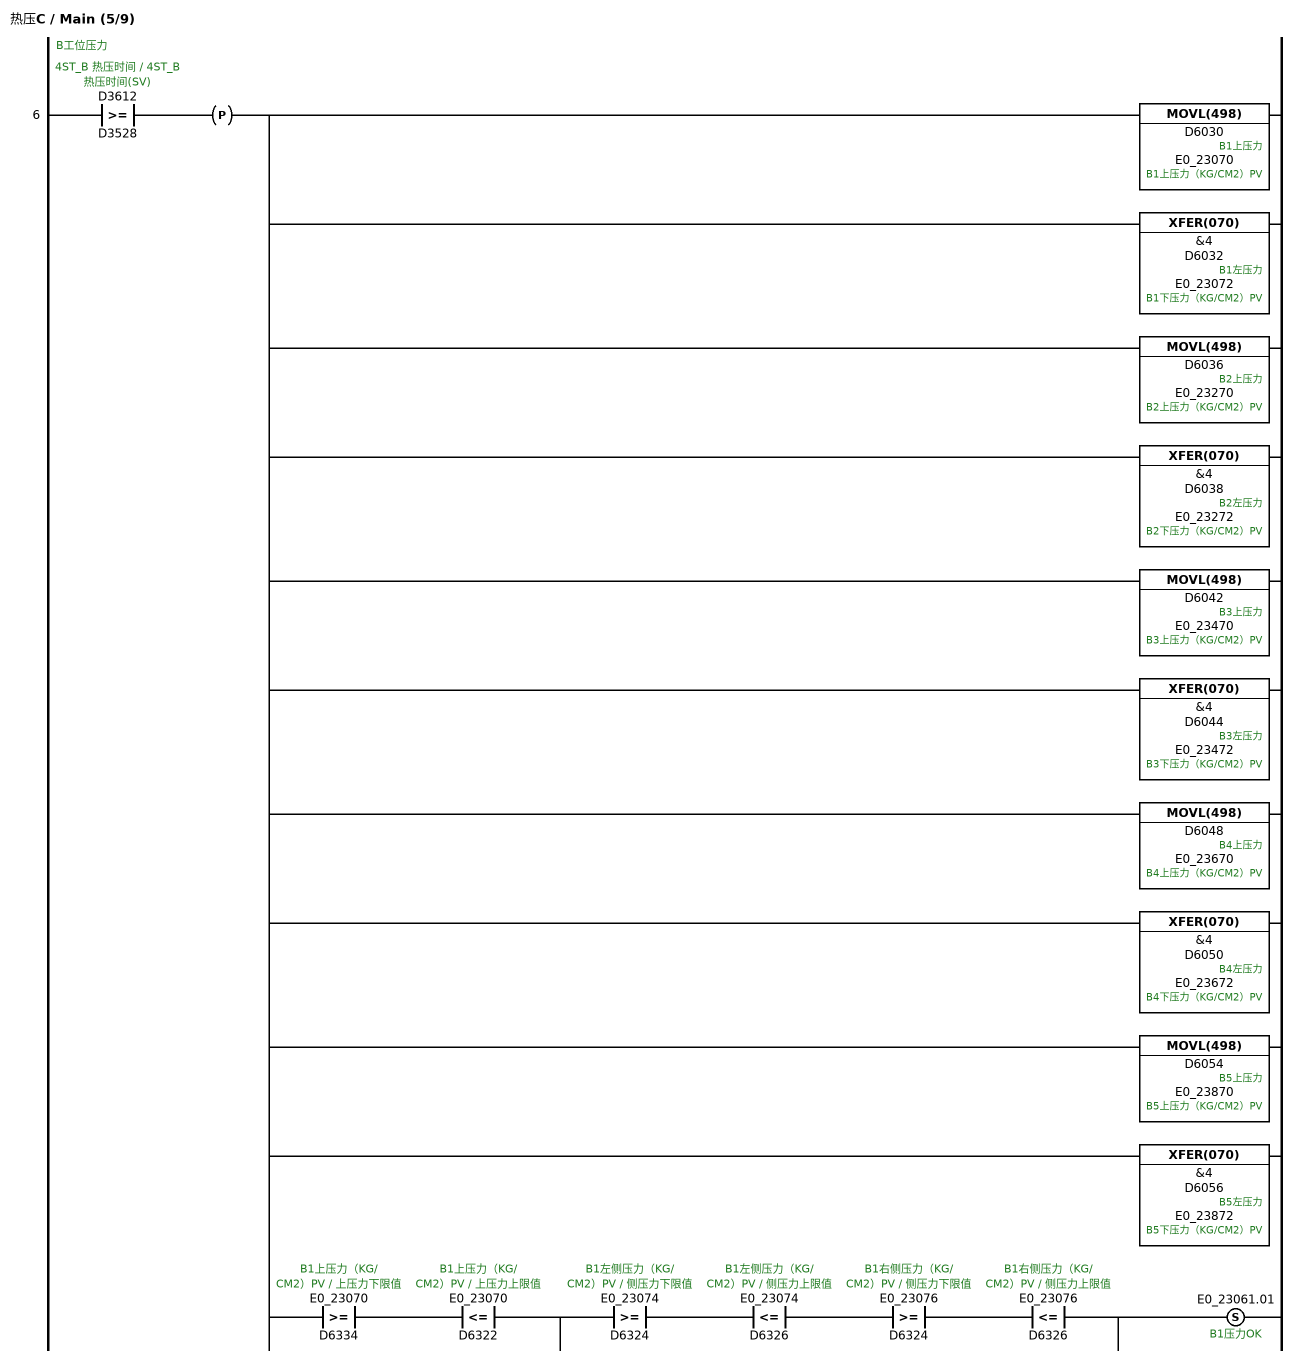

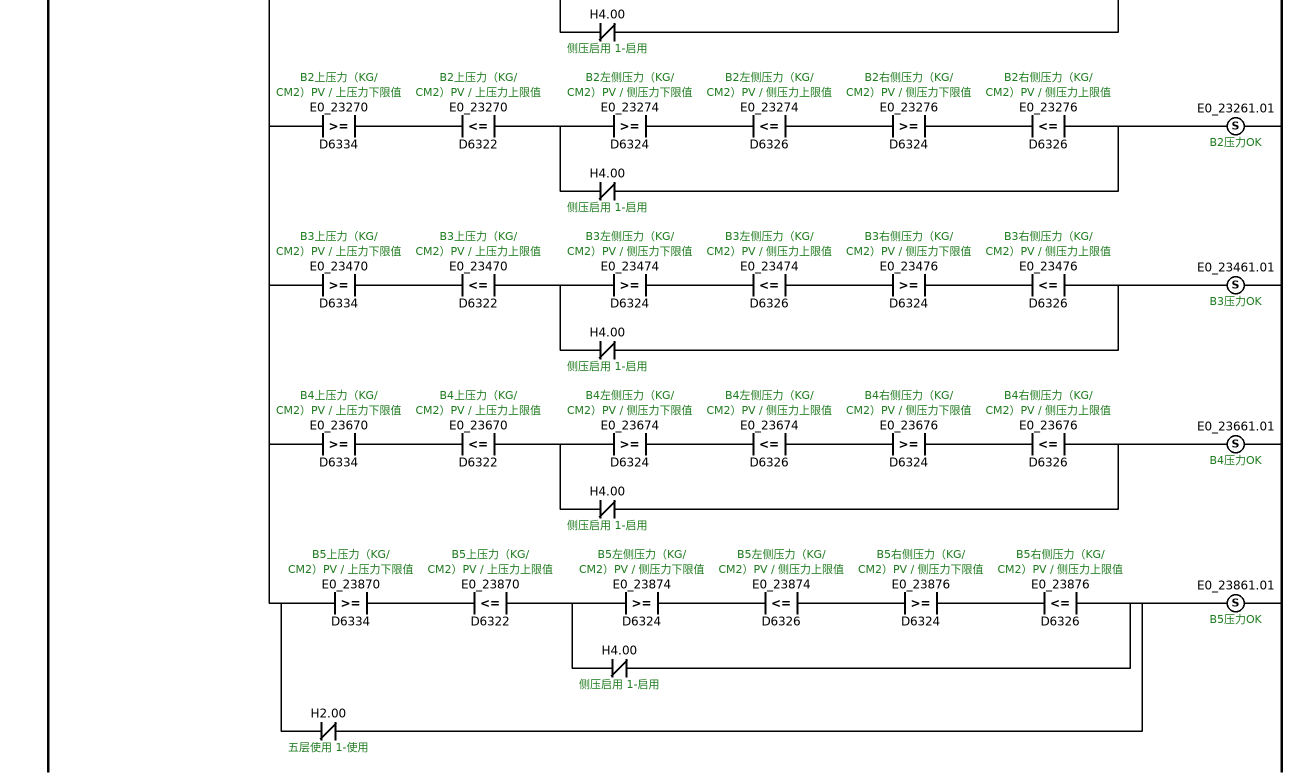
; rung 6: B工位压力
LD>=(325) D3612 D3528  ; 4ST_B 热压时间, 4ST_B 热压时间(SV)
UP(521)
OUT TR0
MOVL(498) D6030 E0_23070  ; B1上压力, B1上压力（KG/CM2）PV
XFER(070) &4 D6032 E0_23072  ; B1左压力, B1下压力（KG/CM2）PV
MOVL(498) D6036 E0_23270  ; B2上压力, B2上压力（KG/CM2）PV
XFER(070) &4 D6038 E0_23272  ; B2左压力, B2下压力（KG/CM2）PV
MOVL(498) D6042 E0_23470  ; B3上压力, B3上压力（KG/CM2）PV
XFER(070) &4 D6044 E0_23472  ; B3左压力, B3下压力（KG/CM2）PV
MOVL(498) D6048 E0_23670  ; B4上压力, B4上压力（KG/CM2）PV
XFER(070) &4 D6050 E0_23672  ; B4左压力, B4下压力（KG/CM2）PV
MOVL(498) D6054 E0_23870  ; B5上压力, B5上压力（KG/CM2）PV
XFER(070) &4 D6056 E0_23872  ; B5左压力, B5下压力（KG/CM2）PV
AND>=L(326) E0_23070 D6334  ; B1上压力（KG/CM2）PV, 上压力下限值
AND<=L(316) E0_23070 D6322  ; B1上压力（KG/CM2）PV, 上压力上限值
LD>=L(326) E0_23074 D6324  ; B1左侧压力（KG/CM2）PV, 侧压力下限值
AND<=L(316) E0_23074 D6326  ; B1左侧压力（KG/CM2）PV, 侧压力上限值
AND>=L(326) E0_23076 D6324  ; B1右侧压力（KG/CM2）PV, 侧压力下限值
AND<=L(316) E0_23076 D6326  ; B1右侧压力（KG/CM2）PV, 侧压力上限值
ORNOT H4.00  ; 侧压启用 1-启用
ANDLD
SET E0_23061.01  ; B1压力OK
LD TR0
AND>=L(326) E0_23270 D6334  ; B2上压力（KG/CM2）PV, 上压力下限值
AND<=L(316) E0_23270 D6322  ; B2上压力（KG/CM2）PV, 上压力上限值
LD>=L(326) E0_23274 D6324  ; B2左侧压力（KG/CM2）PV, 侧压力下限值
AND<=L(316) E0_23274 D6326  ; B2左侧压力（KG/CM2）PV, 侧压力上限值
AND>=L(326) E0_23276 D6324  ; B2右侧压力（KG/CM2）PV, 侧压力下限值
AND<=L(316) E0_23276 D6326  ; B2右侧压力（KG/CM2）PV, 侧压力上限值
ORNOT H4.00  ; 侧压启用 1-启用
ANDLD
SET E0_23261.01  ; B2压力OK
LD TR0
AND>=L(326) E0_23470 D6334  ; B3上压力（KG/CM2）PV, 上压力下限值
AND<=L(316) E0_23470 D6322  ; B3上压力（KG/CM2）PV, 上压力上限值
LD>=L(326) E0_23474 D6324  ; B3左侧压力（KG/CM2）PV, 侧压力下限值
AND<=L(316) E0_23474 D6326  ; B3左侧压力（KG/CM2）PV, 侧压力上限值
AND>=L(326) E0_23476 D6324  ; B3右侧压力（KG/CM2）PV, 侧压力下限值
AND<=L(316) E0_23476 D6326  ; B3右侧压力（KG/CM2）PV, 侧压力上限值
ORNOT H4.00  ; 侧压启用 1-启用
ANDLD
SET E0_23461.01  ; B3压力OK
LD TR0
AND>=L(326) E0_23670 D6334  ; B4上压力（KG/CM2）PV, 上压力下限值
AND<=L(316) E0_23670 D6322  ; B4上压力（KG/CM2）PV, 上压力上限值
LD>=L(326) E0_23674 D6324  ; B4左侧压力（KG/CM2）PV, 侧压力下限值
AND<=L(316) E0_23674 D6326  ; B4左侧压力（KG/CM2）PV, 侧压力上限值
AND>=L(326) E0_23676 D6324  ; B4右侧压力（KG/CM2）PV, 侧压力下限值
AND<=L(316) E0_23676 D6326  ; B4右侧压力（KG/CM2）PV, 侧压力上限值
ORNOT H4.00  ; 侧压启用 1-启用
ANDLD
SET E0_23661.01  ; B4压力OK
LD TR0
LD>=L(326) E0_23870 D6334  ; B5上压力（KG/CM2）PV, 上压力下限值
AND<=L(316) E0_23870 D6322  ; B5上压力（KG/CM2）PV, 上压力上限值
LD>=L(326) E0_23874 D6324  ; B5左侧压力（KG/CM2）PV, 侧压力下限值
AND<=L(316) E0_23874 D6326  ; B5左侧压力（KG/CM2）PV, 侧压力上限值
AND>=L(326) E0_23876 D6324  ; B5右侧压力（KG/CM2）PV, 侧压力下限值
AND<=L(316) E0_23876 D6326  ; B5右侧压力（KG/CM2）PV, 侧压力上限值
ORNOT H4.00  ; 侧压启用 1-启用
ANDLD
ORNOT H2.00  ; 五层使用 1-使用
ANDLD
SET E0_23861.01  ; B5压力OK

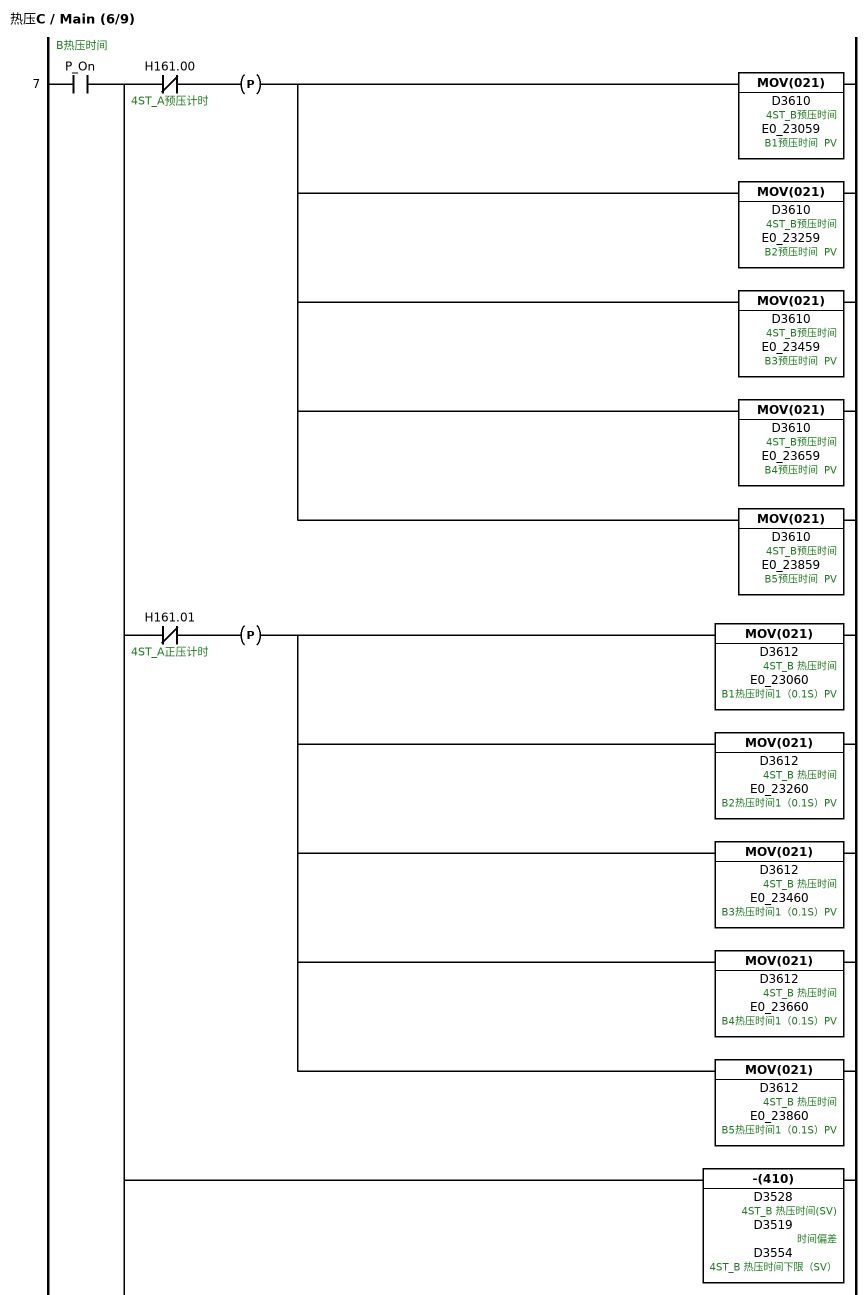

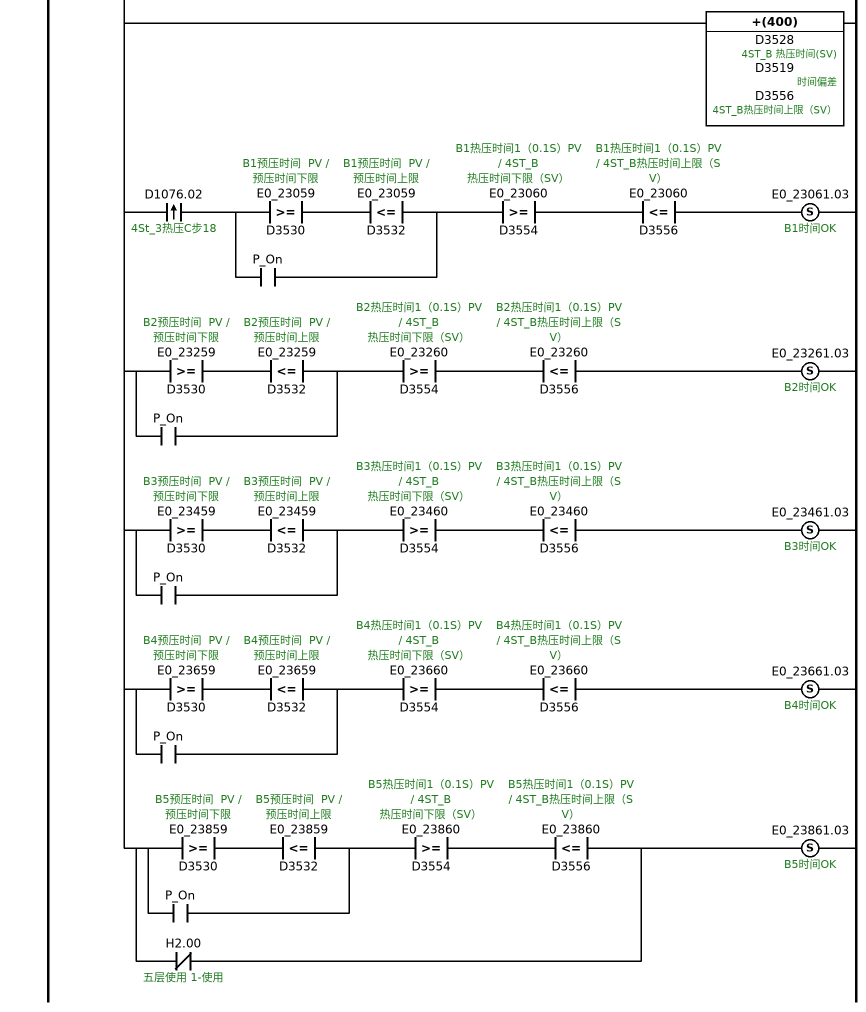
; rung 7: B热压时间
LD P_On
OUT TR0
ANDNOT H161.00  ; 4ST_A预压计时
UP(521)
MOV(021) D3610 E0_23059  ; 4ST_B预压时间, B1预压时间  PV
MOV(021) D3610 E0_23259  ; 4ST_B预压时间, B2预压时间  PV
MOV(021) D3610 E0_23459  ; 4ST_B预压时间, B3预压时间  PV
MOV(021) D3610 E0_23659  ; 4ST_B预压时间, B4预压时间  PV
MOV(021) D3610 E0_23859  ; 4ST_B预压时间, B5预压时间  PV
LD TR0
ANDNOT H161.01  ; 4ST_A正压计时
UP(521)
MOV(021) D3612 E0_23060  ; 4ST_B 热压时间, B1热压时间1（0.1S）PV
MOV(021) D3612 E0_23260  ; 4ST_B 热压时间, B2热压时间1（0.1S）PV
MOV(021) D3612 E0_23460  ; 4ST_B 热压时间, B3热压时间1（0.1S）PV
MOV(021) D3612 E0_23660  ; 4ST_B 热压时间, B4热压时间1（0.1S）PV
MOV(021) D3612 E0_23860  ; 4ST_B 热压时间, B5热压时间1（0.1S）PV
LD TR0
-(410) D3528 D3519 D3554  ; 4ST_B 热压时间(SV), 时间偏差, 4ST_B 热压时间下限（SV）
+(400) D3528 D3519 D3556  ; 4ST_B 热压时间(SV), 时间偏差, 4ST_B热压时间上限（SV）
@AND D1076.02  ; 4St_3热压C步18
LD>=(325) E0_23059 D3530  ; B1预压时间  PV, 预压时间下限
AND<=(315) E0_23059 D3532  ; B1预压时间  PV, 预压时间上限
OR P_On
ANDLD
AND>=(325) E0_23060 D3554  ; B1热压时间1（0.1S）PV, 4ST_B 热压时间下限（SV）
AND<=(315) E0_23060 D3556  ; B1热压时间1（0.1S）PV, 4ST_B热压时间上限（SV）
SET E0_23061.03  ; B1时间OK
LD TR0
LD>=(325) E0_23259 D3530  ; B2预压时间  PV, 预压时间下限
AND<=(315) E0_23259 D3532  ; B2预压时间  PV, 预压时间上限
OR P_On
ANDLD
AND>=(325) E0_23260 D3554  ; B2热压时间1（0.1S）PV, 4ST_B 热压时间下限（SV）
AND<=(315) E0_23260 D3556  ; B2热压时间1（0.1S）PV, 4ST_B热压时间上限（SV）
SET E0_23261.03  ; B2时间OK
LD TR0
LD>=(325) E0_23459 D3530  ; B3预压时间  PV, 预压时间下限
AND<=(315) E0_23459 D3532  ; B3预压时间  PV, 预压时间上限
OR P_On
ANDLD
AND>=(325) E0_23460 D3554  ; B3热压时间1（0.1S）PV, 4ST_B 热压时间下限（SV）
AND<=(315) E0_23460 D3556  ; B3热压时间1（0.1S）PV, 4ST_B热压时间上限（SV）
SET E0_23461.03  ; B3时间OK
LD TR0
LD>=(325) E0_23659 D3530  ; B4预压时间  PV, 预压时间下限
AND<=(315) E0_23659 D3532  ; B4预压时间  PV, 预压时间上限
OR P_On
ANDLD
AND>=(325) E0_23660 D3554  ; B4热压时间1（0.1S）PV, 4ST_B 热压时间下限（SV）
AND<=(315) E0_23660 D3556  ; B4热压时间1（0.1S）PV, 4ST_B热压时间上限（SV）
SET E0_23661.03  ; B4时间OK
LD TR0
LD>=(325) E0_23859 D3530  ; B5预压时间  PV, 预压时间下限
AND<=(315) E0_23859 D3532  ; B5预压时间  PV, 预压时间上限
OR P_On
AND>=(325) E0_23860 D3554  ; B5热压时间1（0.1S）PV, 4ST_B 热压时间下限（SV）
AND<=(315) E0_23860 D3556  ; B5热压时间1（0.1S）PV, 4ST_B热压时间上限（SV）
ORNOT H2.00  ; 五层使用 1-使用
ANDLD
SET E0_23861.03  ; B5时间OK

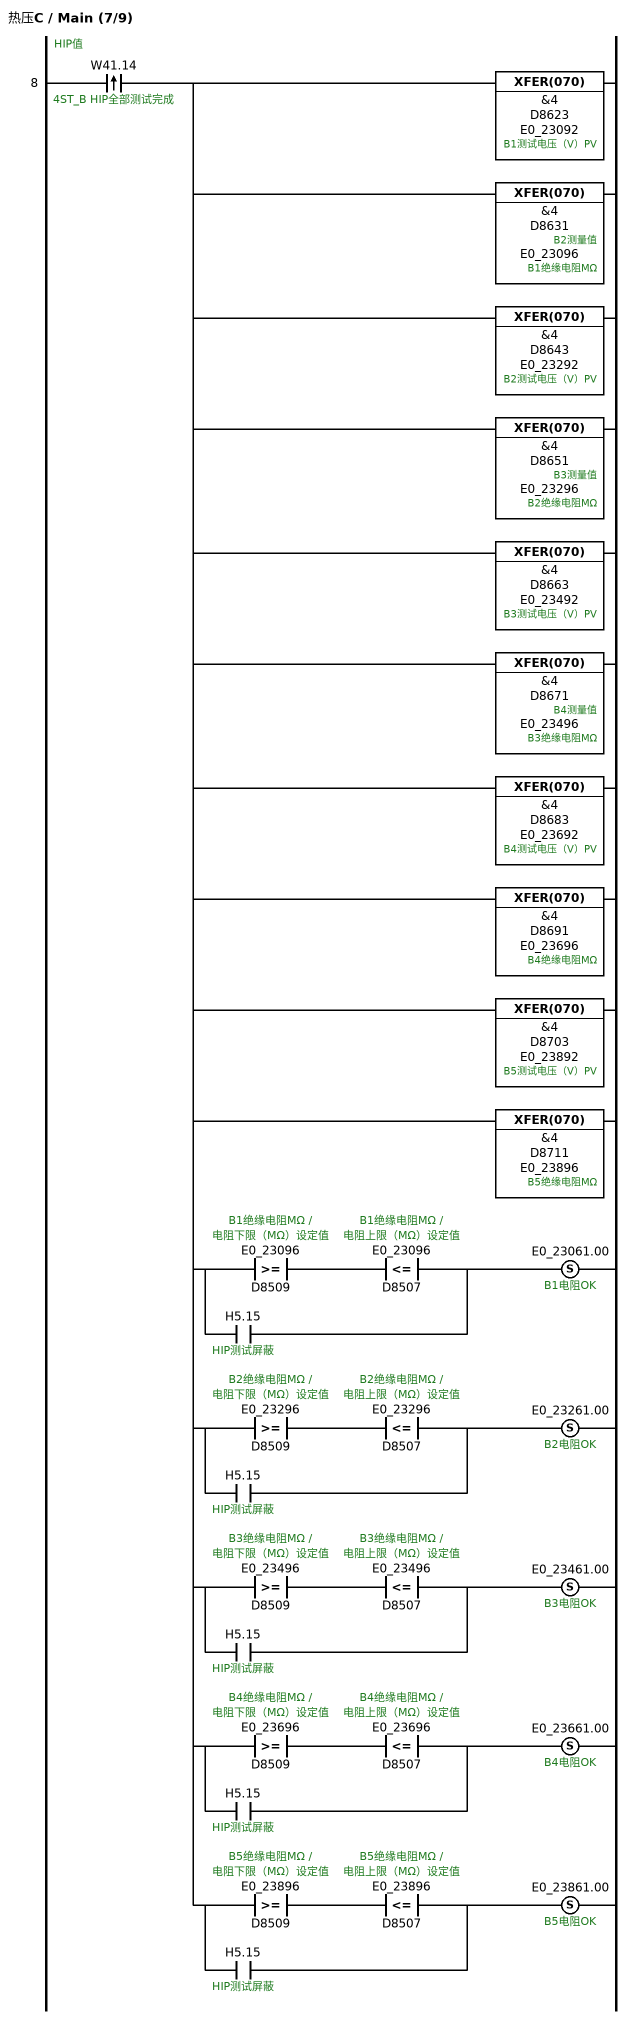
; rung 8: HIP值
@LD W41.14  ; 4ST_B HIP全部测试完成
OUT TR0
XFER(070) &4 D8623 E0_23092  ; B1测试电压（V）PV
XFER(070) &4 D8631 E0_23096  ; B2测量值, B1绝缘电阻MΩ
XFER(070) &4 D8643 E0_23292  ; B2测试电压（V）PV
XFER(070) &4 D8651 E0_23296  ; B3测量值, B2绝缘电阻MΩ
XFER(070) &4 D8663 E0_23492  ; B3测试电压（V）PV
XFER(070) &4 D8671 E0_23496  ; B4测量值, B3绝缘电阻MΩ
XFER(070) &4 D8683 E0_23692  ; B4测试电压（V）PV
XFER(070) &4 D8691 E0_23696  ; B4绝缘电阻MΩ
XFER(070) &4 D8703 E0_23892  ; B5测试电压（V）PV
XFER(070) &4 D8711 E0_23896  ; B5绝缘电阻MΩ
LD>=F(334) E0_23096 D8509  ; B1绝缘电阻MΩ, 电阻下限（MΩ）设定值
AND<=F(332) E0_23096 D8507  ; B1绝缘电阻MΩ, 电阻上限（MΩ）设定值
OR H5.15  ; HIP测试屏蔽
ANDLD
SET E0_23061.00  ; B1电阻OK
LD TR0
LD>=F(334) E0_23296 D8509  ; B2绝缘电阻MΩ, 电阻下限（MΩ）设定值
AND<=F(332) E0_23296 D8507  ; B2绝缘电阻MΩ, 电阻上限（MΩ）设定值
OR H5.15  ; HIP测试屏蔽
ANDLD
SET E0_23261.00  ; B2电阻OK
LD TR0
LD>=F(334) E0_23496 D8509  ; B3绝缘电阻MΩ, 电阻下限（MΩ）设定值
AND<=F(332) E0_23496 D8507  ; B3绝缘电阻MΩ, 电阻上限（MΩ）设定值
OR H5.15  ; HIP测试屏蔽
ANDLD
SET E0_23461.00  ; B3电阻OK
LD TR0
LD>=F(334) E0_23696 D8509  ; B4绝缘电阻MΩ, 电阻下限（MΩ）设定值
AND<=F(332) E0_23696 D8507  ; B4绝缘电阻MΩ, 电阻上限（MΩ）设定值
OR H5.15  ; HIP测试屏蔽
ANDLD
SET E0_23661.00  ; B4电阻OK
LD TR0
LD>=F(334) E0_23896 D8509  ; B5绝缘电阻MΩ, 电阻下限（MΩ）设定值
AND<=F(332) E0_23896 D8507  ; B5绝缘电阻MΩ, 电阻上限（MΩ）设定值
OR H5.15  ; HIP测试屏蔽
ANDLD
SET E0_23861.00  ; B5电阻OK

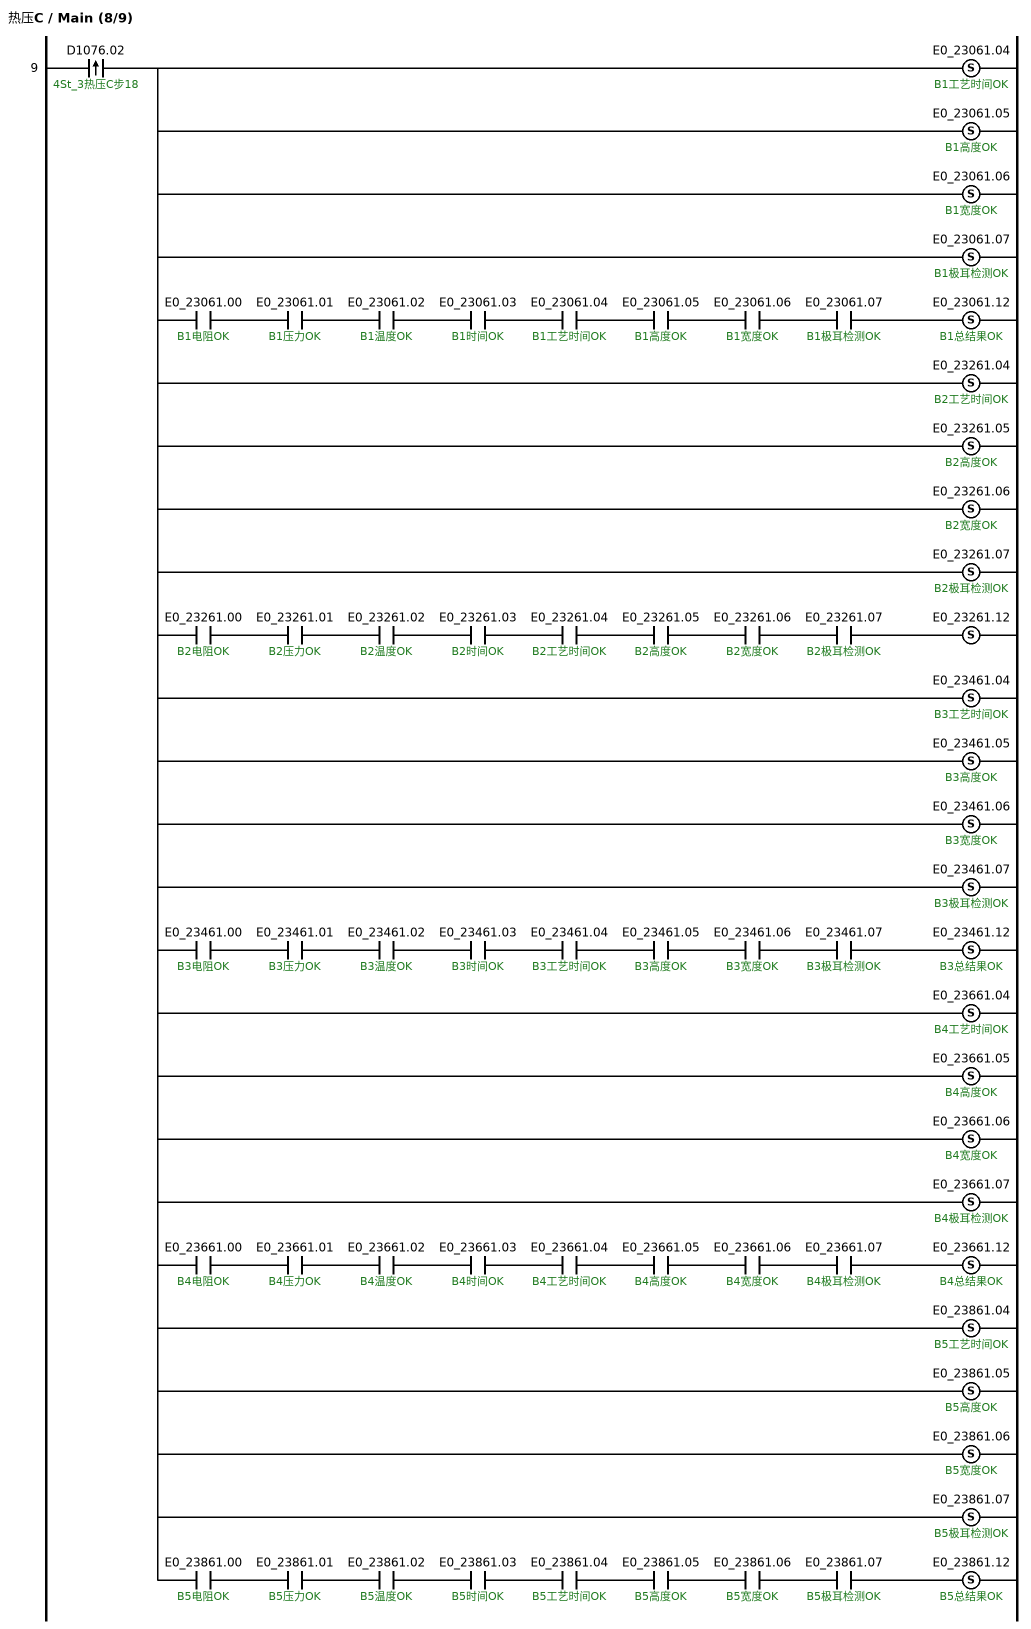
; rung 9
@LD D1076.02  ; 4St_3热压C步18
OUT TR0
SET E0_23061.04  ; B1工艺时间OK
SET E0_23061.05  ; B1高度OK
SET E0_23061.06  ; B1宽度OK
SET E0_23061.07  ; B1极耳检测OK
AND E0_23061.00  ; B1电阻OK
AND E0_23061.01  ; B1压力OK
AND E0_23061.02  ; B1温度OK
AND E0_23061.03  ; B1时间OK
AND E0_23061.04  ; B1工艺时间OK
AND E0_23061.05  ; B1高度OK
AND E0_23061.06  ; B1宽度OK
AND E0_23061.07  ; B1极耳检测OK
SET E0_23061.12  ; B1总结果OK
LD TR0
SET E0_23261.04  ; B2工艺时间OK
SET E0_23261.05  ; B2高度OK
SET E0_23261.06  ; B2宽度OK
SET E0_23261.07  ; B2极耳检测OK
AND E0_23261.00  ; B2电阻OK
AND E0_23261.01  ; B2压力OK
AND E0_23261.02  ; B2温度OK
AND E0_23261.03  ; B2时间OK
AND E0_23261.04  ; B2工艺时间OK
AND E0_23261.05  ; B2高度OK
AND E0_23261.06  ; B2宽度OK
AND E0_23261.07  ; B2极耳检测OK
SET E0_23261.12
LD TR0
SET E0_23461.04  ; B3工艺时间OK
SET E0_23461.05  ; B3高度OK
SET E0_23461.06  ; B3宽度OK
SET E0_23461.07  ; B3极耳检测OK
AND E0_23461.00  ; B3电阻OK
AND E0_23461.01  ; B3压力OK
AND E0_23461.02  ; B3温度OK
AND E0_23461.03  ; B3时间OK
AND E0_23461.04  ; B3工艺时间OK
AND E0_23461.05  ; B3高度OK
AND E0_23461.06  ; B3宽度OK
AND E0_23461.07  ; B3极耳检测OK
SET E0_23461.12  ; B3总结果OK
LD TR0
SET E0_23661.04  ; B4工艺时间OK
SET E0_23661.05  ; B4高度OK
SET E0_23661.06  ; B4宽度OK
SET E0_23661.07  ; B4极耳检测OK
AND E0_23661.00  ; B4电阻OK
AND E0_23661.01  ; B4压力OK
AND E0_23661.02  ; B4温度OK
AND E0_23661.03  ; B4时间OK
AND E0_23661.04  ; B4工艺时间OK
AND E0_23661.05  ; B4高度OK
AND E0_23661.06  ; B4宽度OK
AND E0_23661.07  ; B4极耳检测OK
SET E0_23661.12  ; B4总结果OK
LD TR0
SET E0_23861.04  ; B5工艺时间OK
SET E0_23861.05  ; B5高度OK
SET E0_23861.06  ; B5宽度OK
SET E0_23861.07  ; B5极耳检测OK
AND E0_23861.00  ; B5电阻OK
AND E0_23861.01  ; B5压力OK
AND E0_23861.02  ; B5温度OK
AND E0_23861.03  ; B5时间OK
AND E0_23861.04  ; B5工艺时间OK
AND E0_23861.05  ; B5高度OK
AND E0_23861.06  ; B5宽度OK
AND E0_23861.07  ; B5极耳检测OK
SET E0_23861.12  ; B5总结果OK

